// TIA Portal project "TIA_project" (V17)

(* hardware
DEVICE "S71500/ET200MP station_1"  S7-1500 station
   slot 0: "Rail_0"  Rack  6ES7 590-1***0-0AA0
   slot 1: "PLC_1"  CPU 1512C-1 PN  6ES7 512-1CK00-0AB0  V2.1
      slot 3: "CPU display_1"  6ES7591-1AA00-0AA0
DEVICE "HMI_1"  TP700 Comfort
   slot 0: "TP700 Comfort"  TP700 Comfort  6AV2 124-0GC01-0AX0  14.0.1.0
   slot 1: "HMI_RT_1"  TP700 Comfort  6AV2 124-0GC01-0AX0  14.0.1.0
   slot 5: "HMI_1.IE_CP_1"  PROFINET Interface  14.0.1.0
      slot 1: "PROFINET Interface_1"  PROFINET Interface
         slot 1: "Port_1"  Port
         slot 2: "Port_2"  Port
   slot 7: "HMI_1.MPI/DP_CP_1"  MPI/DP Interface  14.0.1.0
*)

// ===== PLC "PLC_1"  CPU 1512C-1 PN =====

VAR_GLOBAL   // PLC tag table "Default tag table"
   "System_Byte" AT %MB1 : Byte;
   "FirstScan" AT %M1.0 : Bool;
   "DiagStatusUpdate" AT %M1.1 : Bool;
   "AlwaysTRUE" AT %M1.2 : Bool;
   "AlwaysFALSE" AT %M1.3 : Bool;
   "Clock_Byte" AT %MB0 : Byte;
   "Clock_10Hz" AT %M0.0 : Bool;
   "Clock_5Hz" AT %M0.1 : Bool;
   "Clock_2.5Hz" AT %M0.2 : Bool;
   "Clock_2Hz" AT %M0.3 : Bool;
   "Clock_1.25Hz" AT %M0.4 : Bool;
   "Clock_1Hz" AT %M0.5 : Bool;
   "Clock_0.625Hz" AT %M0.6 : Bool;
   "Clock_0.5Hz" AT %M0.7 : Bool;
END_VAR

VAR_GLOBAL   // PLC tag table "IO"
   "diVlaveFill_Open" AT %I320.0 : Bool;
   "diVlaveFill_Close" AT %I320.1 : Bool;
   "diVlaveFill_Error" AT %I320.2 : Bool;
   "diVlaveDrain_Open" AT %I320.3 : Bool;
   "diVlaveDrain_Close" AT %I320.4 : Bool;
   "diVlaveDrain_Error" AT %I320.5 : Bool;
   "diMixer_Run" AT %I320.6 : Bool;
   "diMixer_Error" AT %I320.7 : Bool;
   "doValveFill_Open" AT %Q360.0 : Bool;
   "doValveFill_Close" AT %Q360.1 : Bool;
   "doValveDrain_Open" AT %Q360.2 : Bool;
   "doValveDrain_Close" AT %Q360.3 : Bool;
   "doMixer_Run" AT %Q360.4 : Bool;
   "aiWaterLevel" AT %IW340 : Int;
   "aoHeatPower" AT %QW380 : Int;
   "doHeatingEnable" AT %Q360.5 : Bool;
   "aiWaterTemp" AT %IW342 : Int;
END_VAR

// folder: MAUP

TYPE "Valve"
   STRUCT
      State : Struct
         Open : Bool;
         Closed : Bool;
         OpenOut : Bool;
         CloseOut : Bool;
         Err : Bool;
         StartUpFail : Bool;
         AutCtrl : Bool;
         ManCtrl : Bool;
         MayRun : Bool;
         MayAutoRun : Bool;
         GenErr : Bool;
         StColor : Int;
      END_STRUCT;
      Cmd : Struct
         AutCtrl : Bool;
         ManCtrl : Bool;
         OpenMan : Bool;
         StopMan : Bool;
         CloseMan : Bool;
         Req2OpenAut : Bool;
         Req2CloseAut : Bool;
         ResetSUF : Bool;
      END_STRUCT;
      Param : Struct
         Time2Open : Time := t#3s;
      END_STRUCT;
   END_STRUCT;
END_TYPE

TYPE "Engine"
   STRUCT
      State : Struct
         RT : DInt;
         Run : Bool;
         RunOut : Bool;
         Err : Bool;
         StartUpFail : Bool;
         AutCtrl : Bool;
         ManCtrl : Bool;
         MayRun : Bool;
         MayAutoRun : Bool;
         GenErr : Bool;
         StateInt : Int;
      END_STRUCT;
      Cmd : Struct
         SetRT : DInt := -1;
         AutCtrl : Bool;
         ManCtrl : Bool;
         TurnOnMan : Bool;
         TurnOffMan : Bool;
         Req2RunAutCtrl : Bool;
         ResetSUF : Bool;
      END_STRUCT;
      Param : Struct
         Time2Start : Time := T#3s;
      END_STRUCT;
   END_STRUCT;
END_TYPE

TYPE "Tank"
   STRUCT
      ValveFill : "Valve";
      ValveDrain : "Valve";
      Mixer : "Engine";
      Heater : "Heater";
      Draining : "PhaseDraining";
      Filling : "PhaseFilling";
      Heating : "PhaseHeating";
      Mixing : "PhaseMixing";
      GlobalError : Bool;
      WaterTemp : "AI";
      WaterLevel : "AI";
   END_STRUCT;
END_TYPE

TYPE "PhaseMixing"
   STRUCT
      Cmd : Struct
         StartAut : Bool;
         StopAut : Bool;
         StartMan : Bool;
         StopMan : Bool;
         PauseMan : Bool;
         ResumeMan : Bool;
         ResetDone : Bool;
         AutCtrl : Bool;
         ManCtrl : Bool;
      END_STRUCT;
      State : Struct
         Running : Bool;
         Idle : Bool;
         Paused : Bool;
         Done : Bool;
         AutCtrl : Bool;
         ManCtrl : Bool;
         StateInt : Int;
      END_STRUCT;
      Param : Struct
         TimeSec : Int;
      END_STRUCT;
   END_STRUCT;
END_TYPE

TYPE "PhaseFilling"
   STRUCT
      Cmd : Struct
         StartAut : Bool;
         StopAut : Bool;
         StartMan : Bool;
         StopMan : Bool;
         PauseMan : Bool;
         ResumeMan : Bool;
         ResetDone : Bool;
         AutCtrl : Bool;
         ManCtrl : Bool;
      END_STRUCT;
      State : Struct
         Running : Bool;
         Idle : Bool;
         Paused : Bool;
         Done : Bool;
         AutCtrl : Bool;
         ManCtrl : Bool;
         Stateint : Int;
      END_STRUCT;
      Param : Struct
         FillLevel : Real;
      END_STRUCT;
      WaterLevel : Real;
   END_STRUCT;
END_TYPE

TYPE "PhaseDraining"
   STRUCT
      Cmd : Struct
         StartAut : Bool;
         StopAut : Bool;
         StartMan : Bool;
         StopMan : Bool;
         PauseMan : Bool;
         ResumeMan : Bool;
         ResetDone : Bool;
         AutCtrl : Bool;
         ManCtrl : Bool;
      END_STRUCT;
      State : Struct
         Running : Bool;
         Idle : Bool;
         Paused : Bool;
         Done : Bool;
         AutCtrl : Bool;
         ManCtrl : Bool;
         StateInt : Int;
      END_STRUCT;
      Param : Struct
         DrainLevel : Real;
      END_STRUCT;
      WaterLevel : Real;
   END_STRUCT;
END_TYPE

TYPE "PhaseHeating"
   STRUCT
      Cmd : Struct
         StartAut : Bool;
         StopAut : Bool;
         StartMan : Bool;
         StopMan : Bool;
         PauseMan : Bool;
         ResumeMan : Bool;
         ResetDone : Bool;
         AutCtrl : Bool;
         ManCtrl : Bool;
      END_STRUCT;
      State : Struct
         Running : Bool;
         Idle : Bool;
         Paused : Bool;
         Done : Bool;
         AutCtrl : Bool;
         ManCtrl : Bool;
         StateInt : Int;
      END_STRUCT;
      Param : Struct
         ReqTemp : Real;
      END_STRUCT;
      WaterTemp : Real;
   END_STRUCT;
END_TYPE

TYPE "AI"
   STRUCT
      AIScaled : Real;
      TransducerLoLevel : Int;
      TransducerHiLevel : Int := 27648;
      ScaledValLoLevel : Real;
      ScaledValHiLevel : Real := 100.0;
   END_STRUCT;
END_TYPE

TYPE "Heater"
   STRUCT
      State : Struct
         EnableOut : Bool;
         HeatingOut : Real;
         AutCtrl : Bool;
         ManCtrl : Bool;
         StateInt : Int;
      END_STRUCT;
      Cmd : Struct
         AutCtrl : Bool;
         ManCtrl : Bool;
         TurnOnMan : Bool;
         TurnOffMan : Bool;
         Req2RunAutCtrl : Bool;
      END_STRUCT;
      Param : Struct
         HeatingPowerManual : Real;
         HeatingSetPointAutomat : Real;
      END_STRUCT;
   END_STRUCT;
END_TYPE

TYPE "ProcessControl"
   STRUCT
      Cmd : Struct
         Stop : Bool;
         Start : Bool;
      END_STRUCT;
      State : Struct
         Phase : Int;
      END_STRUCT;
   END_STRUCT;
END_TYPE

// folder: (top level)

DATA_BLOCK "ProcessControlFC_DB"   // DB2
{ S7_Optimized_Access := 'TRUE' }
VERSION : 0.1
// stored: InstanceOfName ProcessControlFC
"ProcessControlFC"
BEGIN
END_DATA_BLOCK

DATA_BLOCK "TankFC_DB"   // DB4
{ S7_Optimized_Access := 'TRUE' }
VERSION : 0.1
// stored: InstanceOfName TankFC
"TankFC"
BEGIN
END_DATA_BLOCK

// folder: DBs

DATA_BLOCK "Data"   // DB1
{ S7_Optimized_Access := 'TRUE' }
VERSION : 0.1
   VAR
      ProcessControl1 : "ProcessControl";
      Tank1 : "Tank";
   END_VAR
BEGIN
   Tank1.Filling.Param.FillLevel := 1.5;
   Tank1.ValveDrain.Param.Time2Open := T#30m;
   Tank1.ValveFill.Param.Time2Open := T#30m;
   Tank1.Mixer.Param.Time2Start := T#30m;
   Tank1.WaterTemp.ScaledValLoLevel := 0.0;
   Tank1.WaterTemp.ScaledValHiLevel := 100.0;
   Tank1.WaterLevel.ScaledValHiLevel := 2.0;
   Tank1.Mixing.Param.TimeSec := 15;
   Tank1.Heating.Param.ReqTemp := 60.0;
   Tank1.Heater.Param.HeatingSetPointAutomat := 60.0;
END_DATA_BLOCK

// folder: (top level)

FUNCTION_BLOCK "TankFC"   // FB3, LAD
{ S7_Optimized_Access := 'TRUE' }
VERSION : 0.1
   VAR_INPUT
      diMixer_Running : Bool;
      diMixer_Error : Bool;
      diValveFill_Open : Bool;
      diValveFill_Close : Bool;
      diValveFill_Error : Bool;
      diValveDrain_Open : Bool;
      diValveDrain_Close : Bool;
      diValveDrain_Error : Bool;
      aiWaterLevel : Int;
      aiWaterTemp : Int;
   END_VAR
   VAR_OUTPUT
      doMixerStart : Bool;
      doValveFill_Open : Bool;
      doValveFill_Close : Bool;
      doValveDrain_Open : Bool;
      doValveDrain_Close : Bool;
      doHeatingEnable : Bool;
      aoReqPowerOfHeating : Word;
   END_VAR
   VAR_IN_OUT
      Tank : "Tank";
   END_VAR
   VAR
      Mixer : "Eng_1DO";
      ValveFill : "Val_2DO";
      ValveDrain : "Val_2DO";
      DrainingFC_Instance : "DrainingFC";
      FillingFC_Instance : "FillingFC";
      MixingFC_Instance : "MixingFC";
      Real2AnalogValue_Instance : "Real2AnalogValue";
      HeatingFC_Instance : "HeatingFC";
      HeaterFC_Instance : "HeaterFC";
   END_VAR
   VAR_TEMP
      HeaterReqPower : Real;
   END_VAR
   VAR_TEMP   // added for the SCL form of the ladder/FBD networks
      _w1 : Bool;
      _w2 : Bool;
   END_VAR
BEGIN

REGION Network 1
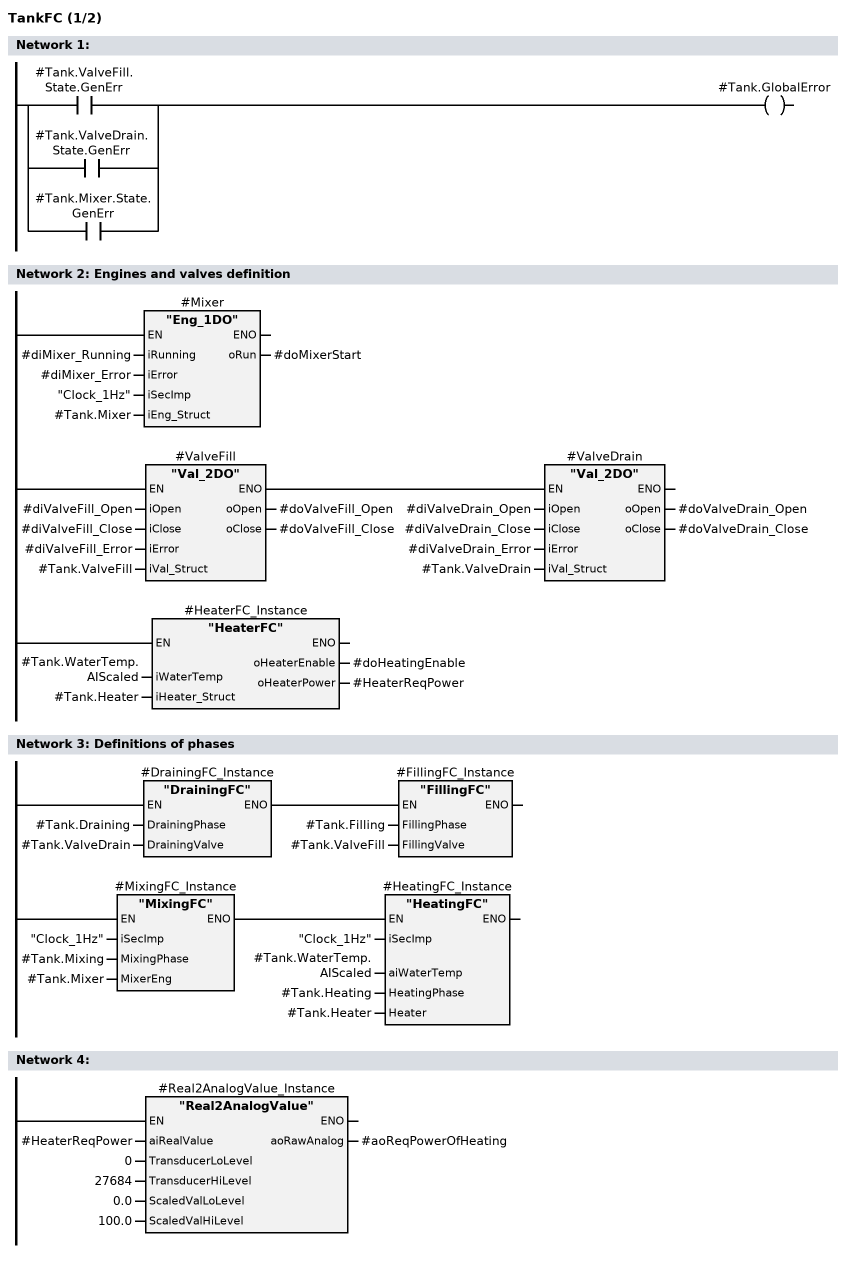
   RUNG wire#powerrail
      Contact( #Tank.ValveFill.State.GenErr )
      wire#w1
      Coil( #Tank.GlobalError )
   END_RUNG
   RUNG wire#powerrail
      Contact( #Tank.ValveDrain.State.GenErr )
   END_RUNG wire#w1
   RUNG wire#powerrail
      Contact( #Tank.Mixer.State.GenErr )
   END_RUNG wire#w1
   // the same network as SCL:
   #Tank.GlobalError := #Tank.ValveFill.State.GenErr OR #Tank.ValveDrain.State.GenErr OR #Tank.Mixer.State.GenErr;
END_REGION

REGION Network 2: Engines and valves definition
   RUNG wire#powerrail
      #Mixer(iRunning := #diMixer_Running, iError := #diMixer_Error, iSecImp := "Clock_1Hz", iEng_Struct := #Tank.Mixer, oRun => #doMixerStart)
   END_RUNG
   RUNG wire#powerrail
      #ValveFill(iOpen := #diValveFill_Open, iClose := #diValveFill_Close, iError := #diValveFill_Error, iVal_Struct := #Tank.ValveFill, oOpen => #doValveFill_Open, oClose => #doValveFill_Close)
      #ValveDrain(iOpen := #diValveDrain_Open, iClose := #diValveDrain_Close, iError := #diValveDrain_Error, iVal_Struct := #Tank.ValveDrain, oOpen => #doValveDrain_Open, oClose => #doValveDrain_Close)
   END_RUNG
   RUNG wire#powerrail
      #HeaterFC_Instance(iWaterTemp := #Tank.WaterTemp.AIScaled, iHeater_Struct := #Tank.Heater, oHeaterEnable => #doHeatingEnable, oHeaterPower => #HeaterReqPower)
   END_RUNG
   // the same network as SCL:
   #Mixer(iRunning := #diMixer_Running,   // "Eng_1DO"
          iError := #diMixer_Error,
          iSecImp := "Clock_1Hz",
          iEng_Struct := #Tank.Mixer,
          oRun => #doMixerStart);
   #ValveFill(iOpen := #diValveFill_Open,   // "Val_2DO"
              iClose := #diValveFill_Close,
              iError := #diValveFill_Error,
              iVal_Struct := #Tank.ValveFill,
              oOpen => #doValveFill_Open,
              oClose => #doValveFill_Close,
              ENO => #_w1);
   IF #_w1 THEN
       #ValveDrain(iOpen := #diValveDrain_Open,   // "Val_2DO"
                   iClose := #diValveDrain_Close,
                   iError := #diValveDrain_Error,
                   iVal_Struct := #Tank.ValveDrain,
                   oOpen => #doValveDrain_Open,
                   oClose => #doValveDrain_Close);
   END_IF;
   #HeaterFC_Instance(iWaterTemp := #Tank.WaterTemp.AIScaled,   // "HeaterFC"
                      iHeater_Struct := #Tank.Heater,
                      oHeaterEnable => #doHeatingEnable,
                      oHeaterPower => #HeaterReqPower);
END_REGION

REGION Network 3: Definitions of phases
   RUNG wire#powerrail
      #DrainingFC_Instance(DrainingPhase := #Tank.Draining, DrainingValve := #Tank.ValveDrain)
      #FillingFC_Instance(FillingPhase := #Tank.Filling, FillingValve := #Tank.ValveFill)
   END_RUNG
   RUNG wire#powerrail
      #MixingFC_Instance(iSecImp := "Clock_1Hz", MixingPhase := #Tank.Mixing, MixerEng := #Tank.Mixer)
      #HeatingFC_Instance(iSecImp := "Clock_1Hz", aiWaterTemp := #Tank.WaterTemp.AIScaled, HeatingPhase := #Tank.Heating, Heater := #Tank.Heater)
   END_RUNG
   // the same network as SCL:
   #DrainingFC_Instance(DrainingPhase := #Tank.Draining, DrainingValve := #Tank.ValveDrain, ENO => #_w1);   // "DrainingFC"
   IF #_w1 THEN
       #FillingFC_Instance(FillingPhase := #Tank.Filling, FillingValve := #Tank.ValveFill);   // "FillingFC"
   END_IF;
   #MixingFC_Instance(iSecImp := "Clock_1Hz", MixingPhase := #Tank.Mixing, MixerEng := #Tank.Mixer, ENO => #_w2);   // "MixingFC"
   IF #_w2 THEN
       #HeatingFC_Instance(iSecImp := "Clock_1Hz",   // "HeatingFC"
                           aiWaterTemp := #Tank.WaterTemp.AIScaled,
                           HeatingPhase := #Tank.Heating,
                           Heater := #Tank.Heater);
   END_IF;
END_REGION

REGION Network 4
   RUNG wire#powerrail
      #Real2AnalogValue_Instance(aiRealValue := #HeaterReqPower, TransducerLoLevel := 0, TransducerHiLevel := 27684, ScaledValLoLevel := 0.0, ScaledValHiLevel := 100.0, aoRawAnalog => #aoReqPowerOfHeating)
   END_RUNG
   // the same network as SCL:
   #Real2AnalogValue_Instance(aiRealValue := #HeaterReqPower,   // "Real2AnalogValue"
                           TransducerLoLevel := 0,
                           TransducerHiLevel := 27684,
                           ScaledValLoLevel := 0.0,
                           ScaledValHiLevel := 100.0,
                           aoRawAnalog => #aoReqPowerOfHeating);
END_REGION

REGION Network 5: Analog scaling
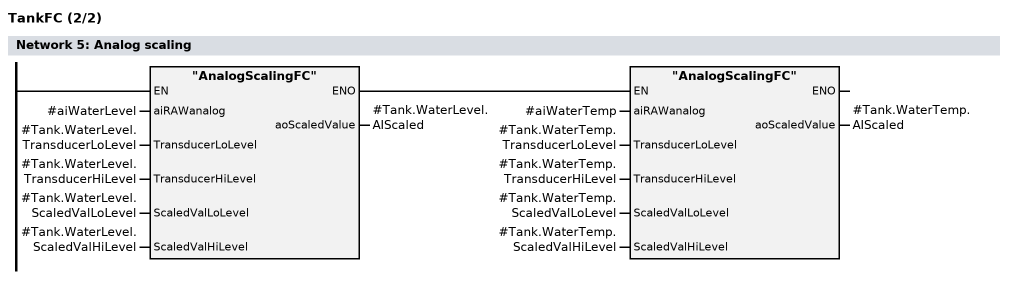
   RUNG wire#powerrail
      "AnalogScalingFC"(aiRAWanalog := #aiWaterLevel, TransducerLoLevel := #Tank.WaterLevel.TransducerLoLevel, TransducerHiLevel := #Tank.WaterLevel.TransducerHiLevel, ScaledValLoLevel := #Tank.WaterLevel.ScaledValLoLevel, ScaledValHiLevel := #Tank.WaterLevel.ScaledValHiLevel, aoScaledValue => #Tank.WaterLevel.AIScaled)
      "AnalogScalingFC"(aiRAWanalog := #aiWaterTemp, TransducerLoLevel := #Tank.WaterTemp.TransducerLoLevel, TransducerHiLevel := #Tank.WaterTemp.TransducerHiLevel, ScaledValLoLevel := #Tank.WaterTemp.ScaledValLoLevel, ScaledValHiLevel := #Tank.WaterTemp.ScaledValHiLevel, aoScaledValue => #Tank.WaterTemp.AIScaled)
   END_RUNG
   // the same network as SCL:
   "AnalogScalingFC"(aiRAWanalog := #aiWaterLevel,
                     TransducerLoLevel := #Tank.WaterLevel.TransducerLoLevel,
                     TransducerHiLevel := #Tank.WaterLevel.TransducerHiLevel,
                     ScaledValLoLevel := #Tank.WaterLevel.ScaledValLoLevel,
                     ScaledValHiLevel := #Tank.WaterLevel.ScaledValHiLevel,
                     aoScaledValue => #Tank.WaterLevel.AIScaled,
                     ENO => #_w1);
   IF #_w1 THEN
       "AnalogScalingFC"(aiRAWanalog := #aiWaterTemp,
                         TransducerLoLevel := #Tank.WaterTemp.TransducerLoLevel,
                         TransducerHiLevel := #Tank.WaterTemp.TransducerHiLevel,
                         ScaledValLoLevel := #Tank.WaterTemp.ScaledValLoLevel,
                         ScaledValHiLevel := #Tank.WaterTemp.ScaledValHiLevel,
                         aoScaledValue => #Tank.WaterTemp.AIScaled);
   END_IF;
END_REGION

REGION Network 6 (SCL): Data transfer
   #Tank.Draining.WaterLevel := #Tank.WaterLevel.AIScaled;
   #Tank.Filling.WaterLevel := #Tank.WaterLevel.AIScaled;
   #Tank.Heating.WaterTemp := #Tank.WaterTemp.AIScaled;
END_REGION
END_FUNCTION_BLOCK

FUNCTION_BLOCK "ProcessControlFC"   // FB10, SCL
{ S7_Optimized_Access := 'TRUE' }
VERSION : 0.1
   VAR_IN_OUT
      Tank : "Tank";
      ProcessControl : "ProcessControl";
   END_VAR
   VAR CONSTANT
      StateIdle : Int := 0;
      StateFilling : Int := 1;
      StateFilled : Int := 2;
      StateHeating : Int := 3;
      StateHeated : Int := 4;
      StateMixing : Int := 5;
      StateMixed : Int := 6;
      StateDraining : Int := 7;
   END_VAR
BEGIN
   CASE #ProcessControl.State.Phase OF
       #StateIdle:
           IF #Tank.Filling.State.Running THEN
               #ProcessControl.State.Phase := #StateFilling;
           END_IF;
       #StateFilling:
           IF #Tank.Filling.State.Done THEN
               #ProcessControl.State.Phase := #StateFilled;
           END_IF;
       #StateFilled:
           #Tank.Heater.Param.HeatingSetPointAutomat := 60;
           #Tank.Mixing.Param.TimeSec := -1;
           #Tank.Heating.Cmd.StartAut := TRUE;
           #Tank.Mixing.Cmd.StartAut := TRUE;
           IF #Tank.Heating.State.Running AND #Tank.Mixing.State.Running THEN
               #ProcessControl.State.Phase := #StateHeating;
           END_IF;
       #StateHeating:
           IF #Tank.Heating.State.Done THEN
               #ProcessControl.State.Phase := #StateHeated;
           END_IF;
       #StateHeated:
           #Tank.Mixing.Param.TimeSec := 30;
           #Tank.Mixing.Cmd.StartAut := TRUE;
           IF #Tank.Mixing.State.Running THEN
               #ProcessControl.State.Phase := #StateMixing;
           END_IF;
       #StateMixing:
           IF #Tank.Mixing.State.Done THEN
               #ProcessControl.State.Phase := #StateMixed;
               #Tank.Heating.Cmd.StopAut := TRUE;
           END_IF;
       #StateMixed:
           #Tank.Draining.Param.DrainLevel := 0;
           #Tank.Draining.Cmd.StartAut := TRUE;
           IF #Tank.Draining.State.Running THEN
               #ProcessControl.State.Phase := #StateDraining;
           END_IF;
       #StateDraining:
           IF #Tank.Draining.#State.Done THEN
               #ProcessControl.State.Phase := #StateIdle;
           END_IF;
   END_CASE;

   IF #ProcessControl.Cmd.Start THEN
       IF #ProcessControl.State.Phase = #StateIdle THEN
           #Tank.Filling.Param.FillLevel := 1.5;
           #Tank.Filling.Cmd.StartAut := TRUE;
       END_IF;
       #ProcessControl.Cmd.Start := FALSE;
   END_IF;

   IF #ProcessControl.Cmd.Stop THEN
       #Tank.Filling.Cmd.StopAut := TRUE;
       #Tank.Heating.Cmd.StopAut := TRUE;
       #Tank.Mixing.Cmd.StopAut := TRUE;
       #Tank.Draining.Cmd.StopAut := TRUE;
       #ProcessControl.State.Phase := #StateIdle;
       #ProcessControl.Cmd.Stop := FALSE;
   END_IF;
END_FUNCTION_BLOCK

ORGANIZATION_BLOCK "Main"   // OB1, LAD, ProgramCycle
TITLE = "Main Program Sweep (Cycle)"
{ S7_Optimized_Access := 'TRUE' }
VERSION : 0.1
   VAR_INPUT
      Initial_Call : Bool;   // Initial call of this OB
      Remanence : Bool;   // =True, if remanent data are available
   END_VAR
BEGIN
END_ORGANIZATION_BLOCK

ORGANIZATION_BLOCK "Cyclic interrupt10ms"   // OB31, LAD, CyclicInterrupt
{ S7_Optimized_Access := 'TRUE' }
VERSION : 0.1
   VAR_INPUT
      Initial_Call : Bool;   // Initial call of this OB
      Event_Count : Int;   // Events discarded
   END_VAR
BEGIN

REGION Network 1
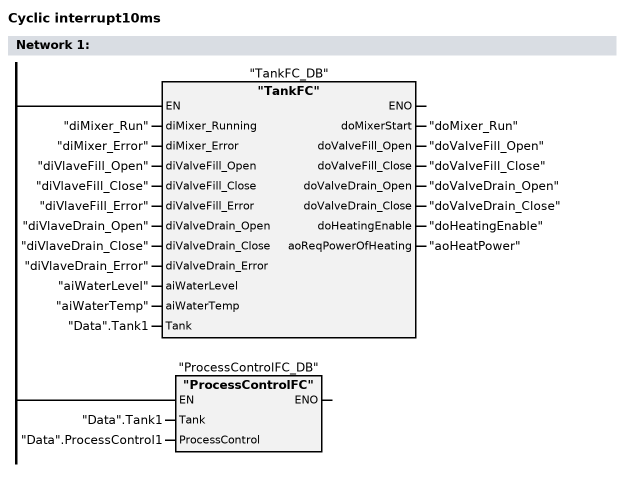
   RUNG wire#powerrail
      "TankFC_DB"(diMixer_Running := "diMixer_Run", diMixer_Error := "diMixer_Error", diValveFill_Open := "diVlaveFill_Open", diValveFill_Close := "diVlaveFill_Close", diValveFill_Error := "diVlaveFill_Error", diValveDrain_Open := "diVlaveDrain_Open", diValveDrain_Close := "diVlaveDrain_Close", diValveDrain_Error := "diVlaveDrain_Error", aiWaterLevel := "aiWaterLevel", aiWaterTemp := "aiWaterTemp", Tank := "Data".Tank1, doMixerStart => "doMixer_Run", doValveFill_Open => "doValveFill_Open", doValveFill_Close => "doValveFill_Close", doValveDrain_Open => "doValveDrain_Open", doValveDrain_Close => "doValveDrain_Close", doHeatingEnable => "doHeatingEnable", aoReqPowerOfHeating => "aoHeatPower")
   END_RUNG
   RUNG wire#powerrail
      "ProcessControlFC_DB"(Tank := "Data".Tank1, ProcessControl := "Data".ProcessControl1)
   END_RUNG
   // the same network as SCL:
   "TankFC_DB"(diMixer_Running := "diMixer_Run",   // "TankFC"
               diMixer_Error := "diMixer_Error",
               diValveFill_Open := "diVlaveFill_Open",
               diValveFill_Close := "diVlaveFill_Close",
               diValveFill_Error := "diVlaveFill_Error",
               diValveDrain_Open := "diVlaveDrain_Open",
               diValveDrain_Close := "diVlaveDrain_Close",
               diValveDrain_Error := "diVlaveDrain_Error",
               aiWaterLevel := "aiWaterLevel",
               aiWaterTemp := "aiWaterTemp",
               Tank := "Data".Tank1,
               doMixerStart => "doMixer_Run",
               doValveFill_Open => "doValveFill_Open",
               doValveFill_Close => "doValveFill_Close",
               doValveDrain_Open => "doValveDrain_Open",
               doValveDrain_Close => "doValveDrain_Close",
               doHeatingEnable => "doHeatingEnable",
               aoReqPowerOfHeating => "aoHeatPower");
   "ProcessControlFC_DB"(Tank := "Data".Tank1, ProcessControl := "Data".ProcessControl1);   // "ProcessControlFC"
END_REGION
END_ORGANIZATION_BLOCK

ORGANIZATION_BLOCK "Startup"   // OB100, SCL, Startup
TITLE = "Complete Restart"
{ S7_Optimized_Access := 'TRUE' }
VERSION : 0.1
   VAR_INPUT
      LostRetentive : Bool;   // True if retentive data are lost
      LostRTC : Bool;   // True if date and time are lost
   END_VAR
BEGIN
END_ORGANIZATION_BLOCK

// folder: FCs

FUNCTION_BLOCK "Eng_1DO"   // FB1, SCL
{ S7_Optimized_Access := 'TRUE' }
VERSION : 0.1
   VAR_INPUT
      iRunning : Bool;
      iError : Bool;
      iSecImp : Bool;
   END_VAR
   VAR_OUTPUT
      oRun : Bool;
   END_VAR
   VAR_IN_OUT
      iEng_Struct : "Engine";
   END_VAR
   VAR
      SecImpEdge : R_TRIG;
      SUF_Timer : TON_TIME;
   END_VAR
   VAR CONSTANT
      Running : Int := 0;
      Stop : Int := 1;
      RunningAndErr : Int := 2;
      Err : Int := 3;
   END_VAR
BEGIN
   REGION RunningTime
       // counting running time of engine - (motoseconds in real situation it should be moto hours)
       // detection rising edge of input secimp - should be conected 1Hz internal clock from PLC

       #SecImpEdge(CLK := #iSecImp);
       IF #SecImpEdge.Q AND #iRunning THEN
           #iEng_Struct.State.RT += 1;
       END_IF;

       IF #iEng_Struct.Cmd.SetRT >= 0 THEN
           #iEng_Struct.State.RT := #iEng_Struct.Cmd.SetRT;
           #iEng_Struct.Cmd.SetRT := -1;
       END_IF;
   END_REGION

   REGION RunState 
       // set real state of engine input into engine structure - input of running
       // engine can be taken from frequential converter, speed sensor, or just
       // from switching element

       #iEng_Struct.State.Run := #iRunning;
   END_REGION

   REGION Manual/Automat 
       // switching state of engine - automatic or manual control (default state is manual)

       IF (#iEng_Struct.Cmd.AutCtrl AND #iEng_Struct.Cmd.ManCtrl) OR (NOT #iEng_Struct.State.AutCtrl AND NOT #iEng_Struct.State.ManCtrl) THEN
           #iEng_Struct.State.AutCtrl := FALSE;
           #iEng_Struct.State.ManCtrl := TRUE;
       ELSIF #iEng_Struct.Cmd.AutCtrl THEN
           #iEng_Struct.State.AutCtrl := TRUE;
           #iEng_Struct.State.ManCtrl := FALSE;
       ELSIF #iEng_Struct.Cmd.ManCtrl THEN
           #iEng_Struct.State.AutCtrl := FALSE;
           #iEng_Struct.State.ManCtrl := TRUE;
       END_IF;

       #iEng_Struct.Cmd.AutCtrl := FALSE;
       #iEng_Struct.Cmd.ManCtrl := FALSE;
   END_REGION

   REGION MR/MAR 
       // setting auxilary signals (may run, may auto run) - MR AND NOT MAR - eng should be started in manual mode,
       // MAR - should be started in automatic mode

       #iEng_Struct.State.MayRun := #iEng_Struct.State.ManCtrl AND NOT #iEng_Struct.State.Err;
       #iEng_Struct.State.MayAutoRun := #iEng_Struct.State.AutCtrl AND NOT #iEng_Struct.State.Err;
   END_REGION

   REGION ManCtrl
       // processing manual actions - if command is processed, it is set to FALSE even if can't be processed
       // Engine commands are turn off (stop) and turn on (start)

       IF #iEng_Struct.Cmd.TurnOnMan AND #iEng_Struct.State.MayRun THEN
           #iEng_Struct.State.RunOut := TRUE;
       END_IF;

       IF #iEng_Struct.Cmd.TurnOffMan AND #iEng_Struct.State.MayRun THEN
           #iEng_Struct.State.RunOut := FALSE;
       END_IF;

       #iEng_Struct.Cmd.TurnOnMan := FALSE;
       #iEng_Struct.Cmd.TurnOffMan := FALSE;
   END_REGION

   REGION AutCtrl 
       //if request to run in automatic mode set outputs to right states if MAR
       //AutoRequest shouldn't be reseted to false state

       IF  #iEng_Struct.State.MayAutoRun THEN
           #iEng_Struct.State.RunOut := #iEng_Struct.Cmd.Req2RunAutCtrl;
       END_IF;
   END_REGION

   REGION ErrStates
       // definition of error states 
       // error - input from digital input of plc - fyzical state of engine 
       // calculating start up fail - if output is sets to start engine, it's expected feedback from running signal in defined time, if feedback doesn't show in this time, it should be start up fail error
       // merge of these two error is general error

       #SUF_Timer(IN := #iEng_Struct.State.RunOut,
                  PT := #iEng_Struct.Param.Time2Start);
       IF #SUF_Timer.Q AND NOT #iRunning THEN
           #iEng_Struct.State.StartUpFail := TRUE;
       END_IF;

       #iEng_Struct.State.Err := #iError;

       #iEng_Struct.State.GenErr := #iEng_Struct.State.StartUpFail OR #iEng_Struct.State.Err;

       IF #iEng_Struct.Cmd.ResetSUF THEN
           #iEng_Struct.State.StartUpFail := FALSE;
       END_IF;
       #iEng_Struct.Cmd.ResetSUF := FALSE;

       IF #iEng_Struct.State.GenErr THEN
           #iEng_Struct.State.RunOut := FALSE;
       END_IF;
   END_REGION

   #oRun := #iEng_Struct.State.RunOut;

   REGION StatusInt
       //write combination of states into int value for visualization (engine - combination of running state and error)

       IF NOT #iEng_Struct.State.GenErr THEN
           IF #iEng_Struct.State.Run THEN
               #iEng_Struct.State.StateInt := #Running;
           ELSE
               #iEng_Struct.State.StateInt := #Stop;
           END_IF;
       ELSE
           IF #iEng_Struct.State.Run THEN
               #iEng_Struct.State.StateInt := #RunningAndErr;
           ELSE
               #iEng_Struct.State.StateInt := #Err;
           END_IF;
       END_IF;
   END_REGION
END_FUNCTION_BLOCK

FUNCTION_BLOCK "Val_2DO"   // FB2, SCL
{ S7_Optimized_Access := 'TRUE' }
VERSION : 0.1
   VAR_INPUT
      iOpen : Bool;
      iClose : Bool;
      iError : Bool;
   END_VAR
   VAR_OUTPUT
      oOpen : Bool;
      oClose : Bool;
   END_VAR
   VAR_IN_OUT
      iVal_Struct : "Valve";
   END_VAR
   VAR
      fTimeToOpen : TON_TIME;
      fTimeToClose : TON_TIME;
   END_VAR
   VAR CONSTANT
      Open : Int := 0;
      Closed : Int := 1;
      OpenAndErr : Int := 2;
      ClosedAndErr : Int := 3;
      NotOpenNotClosedNotErr : Int := 4;
      NotOpenNotClosedAndErr : Int := 5;
      OpenAndClosedAndErr : Int := 6;
      OpenAndClosedNotErr : Int := 7;
   END_VAR
BEGIN
   REGION OpenState 
       // set real state of valve input into valve structure - input of valve can be taken from limit sensor...
       // input - open?
       #iVal_Struct.State.Open := #iOpen;
       // input - closed?
       #iVal_Struct.State.Closed := #iClose;
   END_REGION

   REGION Manual/Automat
       // switching state of engine - automatic or manual control (default state is manual)
       IF (#iVal_Struct.Cmd.AutCtrl AND #iVal_Struct.Cmd.ManCtrl) OR (NOT #iVal_Struct.State.AutCtrl AND NOT #iVal_Struct.State.ManCtrl) THEN
           #iVal_Struct.State.AutCtrl := FALSE;
           #iVal_Struct.State.ManCtrl := TRUE;
       ELSIF #iVal_Struct.Cmd.AutCtrl THEN
           #iVal_Struct.State.AutCtrl := TRUE;
           #iVal_Struct.State.ManCtrl := FALSE;
       ELSIF #iVal_Struct.Cmd.ManCtrl THEN
           #iVal_Struct.State.AutCtrl := FALSE;
           #iVal_Struct.State.ManCtrl := TRUE;
       END_IF;

       #iVal_Struct.Cmd.AutCtrl := FALSE;
       #iVal_Struct.Cmd.ManCtrl := FALSE;
   END_REGION

   REGION MR/MAR
       // setting auxilary signals (may run, may auto run) - MR AND NOT MAR - eng should be started in manual mode, MAR - should be started in automatic mode

       #iVal_Struct.State.MayRun := #iVal_Struct.State.ManCtrl AND NOT #iVal_Struct.State.Err;
       #iVal_Struct.State.MayAutoRun := #iVal_Struct.State.AutCtrl AND NOT #iVal_Struct.State.Err;
   END_REGION

   REGION ManCtrl
       // processing manual actions - if command is processed, it is sets to FALSE even if can't be processed
       // Valve commands are open, close and stop - valve can be stopped intermediate position

       // Open control
       IF #iVal_Struct.Cmd.OpenMan AND #iVal_Struct.State.MayRun THEN
           #iVal_Struct.State.CloseOut := FALSE;
           #iVal_Struct.State.OpenOut := TRUE;
       END_IF;

       // Close control
       IF #iVal_Struct.Cmd.CloseMan AND #iVal_Struct.State.MayRun THEN
           #iVal_Struct.State.OpenOut := FALSE;
           #iVal_Struct.State.CloseOut := TRUE;
       END_IF;

       // stop control
       IF #iVal_Struct.Cmd.StopMan AND #iVal_Struct.State.MayRun THEN
           #iVal_Struct.State.OpenOut := FALSE;
           #iVal_Struct.State.CloseOut := FALSE;
       END_IF;

       // clear commands
       #iVal_Struct.Cmd.OpenMan := FALSE;
       #iVal_Struct.Cmd.StopMan := FALSE;
       #iVal_Struct.Cmd.CloseMan := FALSE;
   END_REGION

   REGION AutCtrl
       //if request to run in automatic mode -> set outputs to right states if MAR
       //AutoRequest shouldn't be reseted to false state
       //if request to open and request to close are setted to 1 simultaneously - outputs should be 0.

       IF #iVal_Struct.State.MayAutoRun THEN
           IF (#iVal_Struct.Cmd.Req2OpenAut AND NOT #iVal_Struct.Cmd.Req2CloseAut) THEN
               #iVal_Struct.State.CloseOut := FALSE;
               #iVal_Struct.State.OpenOut := TRUE;
           ELSIF (NOT #iVal_Struct.Cmd.Req2OpenAut AND #iVal_Struct.Cmd.Req2CloseAut) THEN
               #iVal_Struct.State.OpenOut := FALSE;
               #iVal_Struct.State.CloseOut := TRUE;
           ELSE // simultanesly activated or deactivated
               #iVal_Struct.State.OpenOut := FALSE;
               #iVal_Struct.State.CloseOut := FALSE;
           END_IF;
       END_IF;

   END_REGION

   REGION ErrStates
       // definition of error states 
       // error - input from digital input of plc - fyzical state of valve
       // calculating start up fail - if output is sets to open or close, it's expected feedback from limit sensor in defined time, if feedback doesn't show in this time, it should be start up fail error
       // merge of these two error is general error
       // error is both inputs (open and closed) true state

       #fTimeToOpen(IN := #iVal_Struct.State.OpenOut AND NOT #iVal_Struct.State.CloseOut,
                    PT := #iVal_Struct.Param.Time2Open);
       #fTimeToClose(IN := NOT #iVal_Struct.State.OpenOut AND #iVal_Struct.State.CloseOut,
                     PT := #iVal_Struct.Param.Time2Open);

       IF (#fTimeToOpen.Q AND NOT #iOpen) OR (#fTimeToClose.Q AND NOT #iClose) THEN
           #iVal_Struct.State.StartUpFail := TRUE;
       END_IF;

       // set the input Error to state 
       #iVal_Struct.State.Err := #iError;

       // Merge the errors
       #iVal_Struct.State.GenErr := #iVal_Struct.State.StartUpFail OR #iVal_Struct.State.Err;

       // start up fail can be reseted by operator, command resetSUF, resets SUF and engine should be started again
       IF #iVal_Struct.Cmd.ResetSUF THEN
           #iVal_Struct.State.StartUpFail := FALSE;
       END_IF;
       // reset the command
       #iVal_Struct.Cmd.ResetSUF := FALSE;

       // if error state exists outputs should be in stop state
       IF #iVal_Struct.State.GenErr THEN
           #iVal_Struct.State.OpenOut := FALSE;
           #iVal_Struct.State.CloseOut := FALSE;
       END_IF;

   END_REGION

   #oOpen := #iVal_Struct.State.OpenOut;
   #oClose := #iVal_Struct.State.CloseOut;

   REGION StatusInt
       //write combination of states into int value for visualization (valve - combination of open, close state and error)
       IF #iVal_Struct.State.Open AND NOT #iVal_Struct.State.Closed AND NOT #iVal_Struct.State.GenErr THEN
           #iVal_Struct.State.StColor := #Open;
       ELSIF NOT #iVal_Struct.State.Open AND #iVal_Struct.State.Closed AND NOT #iVal_Struct.State.GenErr THEN
           #iVal_Struct.State.StColor := #Closed;
       ELSIF #iVal_Struct.State.Open AND NOT #iVal_Struct.State.Closed AND #iVal_Struct.State.GenErr THEN
           #iVal_Struct.State.StColor := #OpenAndErr;
       ELSIF NOT #iVal_Struct.State.Open AND #iVal_Struct.State.Closed AND #iVal_Struct.State.GenErr THEN
           #iVal_Struct.State.StColor := #ClosedAndErr;
       ELSIF NOT #iVal_Struct.State.Open AND NOT #iVal_Struct.State.Closed AND NOT #iVal_Struct.State.GenErr THEN
           #iVal_Struct.State.StColor := #NotOpenNotClosedNotErr;
       ELSIF NOT #iVal_Struct.State.Open AND NOT #iVal_Struct.State.Closed AND #iVal_Struct.State.GenErr THEN
           #iVal_Struct.State.StColor := #NotOpenNotClosedAndErr;
       ELSIF #iVal_Struct.State.Open AND #iVal_Struct.State.Closed AND #iVal_Struct.State.GenErr THEN
           #iVal_Struct.State.StColor := #OpenAndClosedAndErr;
       ELSIF #iVal_Struct.State.Open AND #iVal_Struct.State.Closed AND NOT #iVal_Struct.State.GenErr THEN
           #iVal_Struct.State.StColor := #OpenAndClosedNotErr;
       END_IF;
   END_REGION
END_FUNCTION_BLOCK

FUNCTION_BLOCK "FillingFC"   // FB4, SCL
{ S7_Optimized_Access := 'TRUE' }
VERSION : 0.1
   VAR_IN_OUT
      FillingPhase : "PhaseFilling";
      FillingValve : "Valve";
   END_VAR
   VAR CONSTANT
      Idle : Int := 0;
      Running : Int := 1;
      Pause : Int := 2;
   END_VAR
BEGIN
   REGION Aut/Man
       // switching state of engine - automatic or manual control (default state is manual)

       IF (#FillingPhase.Cmd.AutCtrl AND #FillingPhase.Cmd.ManCtrl) OR (NOT #FillingPhase.State.AutCtrl AND NOT #FillingPhase.State.ManCtrl) THEN
           #FillingPhase.State.AutCtrl := FALSE;
           #FillingPhase.State.ManCtrl := TRUE;
       ELSIF #FillingPhase.Cmd.AutCtrl THEN
           #FillingPhase.State.AutCtrl := TRUE;
           #FillingPhase.State.ManCtrl := FALSE;
       ELSIF #FillingPhase.Cmd.ManCtrl THEN
           #FillingPhase.State.AutCtrl := FALSE;
           #FillingPhase.State.ManCtrl := TRUE;
       END_IF;

       #FillingPhase.Cmd.AutCtrl := FALSE;
       #FillingPhase.Cmd.ManCtrl := FALSE;
    END_REGION

   REGION ManCtrl
       // processing manual actions - if command is processed, it is sets to FALSE even if can't be processed
       // Phase commands are start, stop, pause and resume 
       // Start - open filling valve 
       // Stop - close filling valve
       // Pause - close filling valve
       // Resume - open filling valve
       // real states of phase are writed into states in phase structure

       IF #FillingPhase.State.ManCtrl THEN
           IF #FillingPhase.Cmd.StartMan AND #FillingPhase.State.Idle THEN
               #FillingPhase.State.Running := TRUE;
               #FillingPhase.State.Idle := FALSE;
               #FillingPhase.State.Paused := FALSE;
               #FillingPhase.State.Done := FALSE;
           ELSIF #FillingPhase.Cmd.StopMan THEN
               #FillingPhase.State.Running := FALSE;
               #FillingPhase.State.Idle := TRUE;
               #FillingPhase.State.Paused := FALSE;
               #FillingPhase.State.Done := FALSE;
           ELSIF #FillingPhase.Cmd.PauseMan AND #FillingPhase.State.Running THEN
               #FillingPhase.State.Running := FALSE;
               #FillingPhase.State.Idle := FALSE;
               #FillingPhase.State.Paused := TRUE;
               #FillingPhase.State.Done := FALSE;
           ELSIF #FillingPhase.Cmd.ResumeMan AND #FillingPhase.State.Paused THEN
               #FillingPhase.State.Running := TRUE;
               #FillingPhase.State.Idle := FALSE;
               #FillingPhase.State.Paused := FALSE;
               #FillingPhase.State.Done := FALSE;
           END_IF;
       END_IF;

       #FillingPhase.Cmd.StartMan := FALSE;
       #FillingPhase.Cmd.StopMan := FALSE;
       #FillingPhase.Cmd.PauseMan := FALSE;
       #FillingPhase.Cmd.ResumeMan := FALSE;
    END_REGION

   REGION AutCtrl
       // if request to run in automatic mode and phase can be run in automatic mode switch phase to running

       IF #FillingPhase.State.AutCtrl THEN
           IF #FillingPhase.Cmd.StartAut THEN
               #FillingPhase.State.Running := TRUE;
               #FillingPhase.State.Idle := FALSE;
               #FillingPhase.State.Paused := FALSE;
               #FillingPhase.State.Done := FALSE;
           ELSIF #FillingPhase.Cmd.StopAut THEN
               #FillingPhase.State.Running := FALSE;
               #FillingPhase.State.Idle := TRUE;
               #FillingPhase.State.Paused := FALSE;
               #FillingPhase.State.Done := FALSE;
           END_IF;
       END_IF;

       #FillingPhase.Cmd.StartAut := FALSE;
       #FillingPhase.Cmd.StopAut := FALSE;
    END_REGION

   REGION Done
       //every phase should have finish condition - filling phase - if water level is above requested level
       //after that done state should be setted to 1

       IF #FillingPhase.State.Running AND (#FillingPhase.WaterLevel >= #FillingPhase.Param.FillLevel AND NOT (#FillingPhase.WaterLevel = 2.0)) THEN
           #FillingPhase.Cmd.StopAut := TRUE;
           #FillingPhase.Cmd.StopMan := TRUE;
           #FillingPhase.State.Done := TRUE;
       END_IF;

       IF #FillingPhase.State.Paused OR #FillingPhase.State.Idle THEN
           #FillingPhase.State.Done := TRUE;
       END_IF;

       // command reset done resets done state and than resets command

       IF #FillingPhase.Cmd.ResetDone THEN
           #FillingPhase.State.Done := FALSE;
       END_IF;
       #FillingPhase.Cmd.ResetDone := FALSE;
   END_REGION

   REGION States 
       //Command valve in cases of states

       IF #FillingPhase.State.Running THEN
           #FillingValve.Cmd.Req2OpenAut := TRUE;
           #FillingValve.Cmd.Req2CloseAut := FALSE;
       ELSE
           #FillingValve.Cmd.Req2OpenAut := FALSE;
           #FillingValve.Cmd.Req2CloseAut := TRUE;
       END_IF;
   END_REGION

   // delault state of phase - if not any state sets state to idle

   IF NOT #FillingPhase.State.Running AND NOT #FillingPhase.State.Idle AND NOT #FillingPhase.State.Paused THEN
       #FillingPhase.State.Idle := TRUE;
   END_IF;

   // write binary states into int value for visualization

   IF #FillingPhase.State.Running THEN
       #FillingPhase.State.Stateint := #Running;
   ELSIF #FillingPhase.State.Idle THEN
       #FillingPhase.State.Stateint := #Idle;
   ELSE
       #FillingPhase.State.Stateint := #Pause;
   END_IF;
END_FUNCTION_BLOCK

FUNCTION_BLOCK "DrainingFC"   // FB5, SCL
{ S7_Optimized_Access := 'TRUE' }
VERSION : 0.1
   VAR_IN_OUT
      DrainingPhase : "PhaseDraining";
      DrainingValve : "Valve";
   END_VAR
   VAR CONSTANT
      Idle : Int := 0;
      Running : Int := 1;
      Pause : Int := 2;
   END_VAR
BEGIN
   REGION Aut/Man
       // switching state of engine - automatic or manual control (default state is manual)

       IF (#DrainingPhase.Cmd.AutCtrl AND #DrainingPhase.Cmd.ManCtrl) OR (NOT #DrainingPhase.State.AutCtrl AND NOT #DrainingPhase.State.ManCtrl) THEN
           #DrainingPhase.State.AutCtrl := FALSE;
           #DrainingPhase.State.ManCtrl := TRUE;
       ELSIF #DrainingPhase.Cmd.AutCtrl THEN
           #DrainingPhase.State.AutCtrl := TRUE;
           #DrainingPhase.State.ManCtrl := FALSE;
       ELSIF #DrainingPhase.Cmd.ManCtrl THEN
           #DrainingPhase.State.AutCtrl := FALSE;
           #DrainingPhase.State.ManCtrl := TRUE;
       END_IF;

       #DrainingPhase.Cmd.AutCtrl := FALSE;
       #DrainingPhase.Cmd.ManCtrl := FALSE;
   END_REGION

   REGION ManCtrl
       // processing manual actions - if command is processed, it is sets to FALSE even if can't be processed
       // Phase commands are start, stop, pause and resume 
       // Start - open draining valve 
       // Stop - close draining valve
       // Pause - close draining valve
       // Resume - open draining valve
       // real states of phase are writed into states in phase structure

       IF #DrainingPhase.State.ManCtrl THEN
           IF #DrainingPhase.Cmd.StartMan AND #DrainingPhase.State.Idle THEN
               #DrainingPhase.State.Running := TRUE;
               #DrainingPhase.State.Idle := FALSE;
               #DrainingPhase.State.Paused := FALSE;
               #DrainingPhase.State.Done := FALSE;
           ELSIF #DrainingPhase.Cmd.StopMan THEN
               #DrainingPhase.State.Running := FALSE;
               #DrainingPhase.State.Idle := TRUE;
               #DrainingPhase.State.Paused := FALSE;
               #DrainingPhase.State.Done := FALSE;
           ELSIF #DrainingPhase.Cmd.PauseMan AND #DrainingPhase.State.Running THEN
               #DrainingPhase.State.Running := FALSE;
               #DrainingPhase.State.Idle := FALSE;
               #DrainingPhase.State.Paused := TRUE;
               #DrainingPhase.State.Done := FALSE;
           ELSIF #DrainingPhase.Cmd.ResumeMan AND #DrainingPhase.State.Paused THEN
               #DrainingPhase.State.Running := TRUE;
               #DrainingPhase.State.Idle := FALSE;
               #DrainingPhase.State.Paused := FALSE;
               #DrainingPhase.State.Done := FALSE;
           END_IF;
       END_IF;

       #DrainingPhase.Cmd.StartMan := FALSE;
       #DrainingPhase.Cmd.StopMan := FALSE;
       #DrainingPhase.Cmd.PauseMan := FALSE;
       #DrainingPhase.Cmd.ResumeMan := FALSE;
   END_REGION

   REGION AutCtrl
       //if request to run in automatic mode -> set auto request to open of filling valve to 1 and close to 0, if not open 0 close 1
       // commands should be sets to false after their processing

       IF #DrainingPhase.State.AutCtrl THEN
           IF #DrainingPhase.Cmd.StartAut THEN
               #DrainingPhase.State.Running := TRUE;
               #DrainingPhase.State.Idle := FALSE;
               #DrainingPhase.State.Paused := FALSE;
               #DrainingPhase.State.Done := FALSE;
           ELSIF #DrainingPhase.Cmd.StopAut THEN
               #DrainingPhase.State.Running := FALSE;
               #DrainingPhase.State.Idle := TRUE;
               #DrainingPhase.State.Paused := FALSE;
               #DrainingPhase.State.Done := FALSE;
           END_IF;
       END_IF;

       #DrainingPhase.Cmd.StartAut := FALSE;
       #DrainingPhase.Cmd.StopAut := FALSE;
   END_REGION

   REGION Done
       //every phase should have finish condition - draining phase - if water level is below requested level
       //after that done state should be setted to 1

       IF #DrainingPhase.State.Running AND (#DrainingPhase.WaterLevel <= #DrainingPhase.Param.DrainLevel OR #DrainingPhase.WaterLevel = 2.0) THEN
           #DrainingPhase.Cmd.StopAut := TRUE;
           #DrainingPhase.Cmd.StopMan := TRUE;
           #DrainingPhase.State.Done := TRUE;
       END_IF;

       IF #DrainingPhase.State.Paused OR #DrainingPhase.State.Idle THEN
           #DrainingPhase.State.Done := TRUE;
       END_IF;

       // command reset done resets done state and than resets command

       IF #DrainingPhase.Cmd.ResetDone THEN
           #DrainingPhase.State.Done := FALSE;
       END_IF;
       #DrainingPhase.Cmd.ResetDone := FALSE;
   END_REGION

   REGION States 
       //Command valve in cases of states

       IF #DrainingPhase.State.Running THEN
           #DrainingValve.Cmd.Req2OpenAut := TRUE;
           #DrainingValve.Cmd.Req2CloseAut := FALSE;
       ELSE
           #DrainingValve.Cmd.Req2OpenAut := FALSE;
           #DrainingValve.Cmd.Req2CloseAut := TRUE;
       END_IF;
   END_REGION

   // delault state of phase - if not any state sets state to idle

   IF NOT #DrainingPhase.State.Running AND NOT #DrainingPhase.State.Idle AND NOT #DrainingPhase.State.Paused THEN
       #DrainingPhase.State.Idle := TRUE;
   END_IF;

   // write binary states into int value for visualization

   IF #DrainingPhase.State.Running THEN
       #DrainingPhase.State.StateInt := #Running;
   ELSIF #DrainingPhase.State.Idle THEN
       #DrainingPhase.State.StateInt := #Idle;
   ELSE
       #DrainingPhase.State.StateInt := #Pause;
   END_IF;
END_FUNCTION_BLOCK

FUNCTION_BLOCK "MixingFC"   // FB6, SCL
{ S7_Optimized_Access := 'TRUE' }
VERSION : 0.1
   VAR_INPUT
      iSecImp : Bool;
   END_VAR
   VAR_IN_OUT
      MixingPhase : "PhaseMixing";
      MixerEng : "Engine";
   END_VAR
   VAR
      fElapsedTime : Int;
      fSecImp : R_TRIG;
   END_VAR
   VAR CONSTANT
      Idle : Int := 0;
      Running : Int := 1;
      Pause : Int := 2;
   END_VAR
BEGIN
   REGION Aut/Man
       // switching state of engine - automatic or manual control (default state is manual)

       IF (#MixingPhase.Cmd.AutCtrl AND #MixingPhase.Cmd.ManCtrl) OR (NOT #MixingPhase.State.AutCtrl AND NOT #MixingPhase.State.ManCtrl) THEN
           #MixingPhase.State.AutCtrl := FALSE;
           #MixingPhase.State.ManCtrl := TRUE;
       ELSIF #MixingPhase.Cmd.AutCtrl THEN
           #MixingPhase.State.AutCtrl := TRUE;
           #MixingPhase.State.ManCtrl := FALSE;
       ELSIF #MixingPhase.Cmd.ManCtrl THEN
           #MixingPhase.State.AutCtrl := FALSE;
           #MixingPhase.State.ManCtrl := TRUE;
       END_IF;

       #MixingPhase.Cmd.AutCtrl := FALSE;
       #MixingPhase.Cmd.ManCtrl := FALSE;
   END_REGION

   REGION ManCtrl
       // processing manual actions - if command is processed, it is sets to FALSE even if can't be processed
       // Phase commands are start, stop, pause and resume 
       // Start - start mixing  
       // Stop - stop mixing
       // Pause - stop mixing 
       // Resume - start mixing
       // real states of phase are writed into states in phase structure

       IF #MixingPhase.State.ManCtrl THEN
           IF #MixingPhase.Cmd.StartMan AND #MixingPhase.State.Idle THEN
               #MixingPhase.State.Running := TRUE;
               #MixingPhase.State.Idle := FALSE;
               #MixingPhase.State.Paused := FALSE;
               #MixingPhase.State.Done := FALSE;
           ELSIF #MixingPhase.Cmd.StopMan THEN
               #MixingPhase.State.Running := FALSE;
               #MixingPhase.State.Idle := TRUE;
               #MixingPhase.State.Paused := FALSE;
               #MixingPhase.State.Done := FALSE;
               #fElapsedTime := 0;
           ELSIF #MixingPhase.Cmd.PauseMan AND #MixingPhase.State.Running THEN
               #MixingPhase.State.Running := FALSE;
               #MixingPhase.State.Idle := FALSE;
               #MixingPhase.State.Paused := TRUE;
               #MixingPhase.State.Done := FALSE;
           ELSIF #MixingPhase.Cmd.ResumeMan AND #MixingPhase.State.Paused THEN
               #MixingPhase.State.Running := TRUE;
               #MixingPhase.State.Idle := FALSE;
               #MixingPhase.State.Paused := FALSE;
               #MixingPhase.State.Done := FALSE;
           END_IF;
       END_IF;

       #MixingPhase.Cmd.StartMan := FALSE;
       #MixingPhase.Cmd.StopMan := FALSE;
       #MixingPhase.Cmd.PauseMan := FALSE;
       #MixingPhase.Cmd.ResumeMan := FALSE;
   END_REGION

   REGION AutCtrl
       // if request to run in automatic mode -> set auto request to mixing to 1, if not request to mixing is 0
       // commands should be sets to false after their processing

       IF #MixingPhase.State.AutCtrl THEN
           IF #MixingPhase.Cmd.StartAut THEN
               #MixingPhase.State.Running := TRUE;
               #MixingPhase.State.Idle := FALSE;
               #MixingPhase.State.Paused := FALSE;
               #MixingPhase.State.Done := FALSE;
           ELSIF #MixingPhase.Cmd.StopAut THEN
               #MixingPhase.State.Running := FALSE;
               #MixingPhase.State.Idle := TRUE;
               #MixingPhase.State.Paused := FALSE;
               #MixingPhase.State.Done := FALSE;
               #fElapsedTime := 0;
           END_IF;
       END_IF;

       #MixingPhase.Cmd.StartAut := FALSE;
       #MixingPhase.Cmd.StopAut := FALSE;
   END_REGION


   REGION Done
       // every phase should have finish condition - mixing phase - if time of runnig is bigger or same as requested
       // after that done state should be setted to 1

       #fSecImp(CLK := #iSecImp);
       IF #fSecImp.Q AND #MixingPhase.State.Running AND NOT (#MixingPhase.Param.TimeSec = -1) THEN
           #fElapsedTime += 1;
       END_IF;

       IF #MixingPhase.State.Running AND #fElapsedTime >= #MixingPhase.Param.TimeSec AND NOT (#MixingPhase.Param.TimeSec = -1) THEN
           #MixingPhase.Cmd.StopAut := TRUE;
           #MixingPhase.Cmd.StopMan := TRUE;
           #MixingPhase.State.Done := TRUE;
       END_IF;

       IF #MixingPhase.State.Paused OR #MixingPhase.State.Idle THEN
           #MixingPhase.State.Done := TRUE;
       END_IF;

       // command reset done resets done state and than resets command

       IF #MixingPhase.Cmd.ResetDone THEN
           #MixingPhase.State.Done := FALSE;
       END_IF;
       #MixingPhase.Cmd.ResetDone := FALSE;
   END_REGION

   REGION States 
       //Command mixer in cases of states

       IF #MixingPhase.State.Running THEN
           #MixerEng.Cmd.Req2RunAutCtrl := TRUE;
       ELSE
           #MixerEng.Cmd.Req2RunAutCtrl := FALSE;
       END_IF;
   END_REGION

   // delault state of phase - if not any state sets state to idle

   IF NOT #MixingPhase.State.Running AND NOT #MixingPhase.State.Idle AND NOT #MixingPhase.State.Paused THEN
       #MixingPhase.State.Idle := TRUE;
   END_IF;

   // write binary states into int value for visualization

   IF #MixingPhase.State.Running THEN
       #MixingPhase.State.StateInt := #Running;
   ELSIF #MixingPhase.State.Idle THEN
       #MixingPhase.State.StateInt := #Idle;
   ELSE
       #MixingPhase.State.StateInt := #Pause;
   END_IF;
END_FUNCTION_BLOCK

FUNCTION_BLOCK "HeaterFC"   // FB7, SCL
{ S7_Optimized_Access := 'TRUE' }
VERSION : 0.1
   VAR_INPUT
      iWaterTemp : Real;
   END_VAR
   VAR_OUTPUT
      oHeaterEnable : Bool;
      oHeaterPower : Real;
   END_VAR
   VAR_IN_OUT
      iHeater_Struct : "Heater";
   END_VAR
   VAR
      fMode : Int;
   END_VAR
BEGIN
   #fMode := 3; // automatic mode of PID component
   "HeatingPID"(Setpoint := #iHeater_Struct.Param.HeatingSetPointAutomat,
                Input := #iWaterTemp,
                ManualEnable := #iHeater_Struct.State.ManCtrl,
                ManualValue := #iHeater_Struct.Param.HeatingPowerManual,
                OutputHeat => #iHeater_Struct.State.HeatingOut,
                Mode := #fMode);

   REGION Manual/Automat

       IF (#iHeater_Struct.Cmd.AutCtrl AND #iHeater_Struct.Cmd.ManCtrl) OR (NOT #iHeater_Struct.State.AutCtrl AND NOT #iHeater_Struct.State.ManCtrl) THEN
           #iHeater_Struct.State.AutCtrl := FALSE;
           #iHeater_Struct.State.ManCtrl := TRUE;
       ELSIF #iHeater_Struct.Cmd.AutCtrl THEN
           #iHeater_Struct.State.AutCtrl := TRUE;
           #iHeater_Struct.State.ManCtrl := FALSE;
       ELSIF #iHeater_Struct.Cmd.ManCtrl THEN
           #iHeater_Struct.State.AutCtrl := FALSE;
           #iHeater_Struct.State.ManCtrl := TRUE;
       END_IF;

       #iHeater_Struct.Cmd.AutCtrl := FALSE;
       #iHeater_Struct.Cmd.ManCtrl := FALSE;
   END_REGION

   REGION ManCtrl

       IF #iHeater_Struct.Cmd.TurnOnMan AND #iHeater_Struct.State.ManCtrl THEN
           // set the state
           #iHeater_Struct.State.EnableOut := TRUE;
       END_IF;

       IF #iHeater_Struct.Cmd.TurnOffMan AND #iHeater_Struct.State.ManCtrl THEN
           #iHeater_Struct.State.EnableOut := FALSE;
       END_IF;

       #iHeater_Struct.Cmd.TurnOnMan := FALSE;
       #iHeater_Struct.Cmd.TurnOffMan := FALSE;
   END_REGION

   REGION AutCtrl

       IF #iHeater_Struct.State.AutCtrl THEN
           #iHeater_Struct.State.EnableOut := #iHeater_Struct.Cmd.Req2RunAutCtrl;
       END_IF;
   END_REGION

   #oHeaterEnable := #iHeater_Struct.State.EnableOut;
   #oHeaterPower := #iHeater_Struct.State.HeatingOut;
END_FUNCTION_BLOCK

FUNCTION_BLOCK "Real2AnalogValue"   // FB8, SCL
{ S7_Optimized_Access := 'TRUE' }
VERSION : 0.1
   VAR_INPUT
      aiRealValue : Real;
      TransducerLoLevel : Int;
      TransducerHiLevel : Int;
      ScaledValLoLevel : Real;
      ScaledValHiLevel : Real;
   END_VAR
   VAR_OUTPUT
      aoRawAnalog : Int;
   END_VAR
BEGIN
   #aoRawAnalog := REAL_TO_INT(((#TransducerHiLevel - #TransducerLoLevel) / (#ScaledValHiLevel - #ScaledValLoLevel)) * (#aiRealValue - #ScaledValLoLevel) + #TransducerLoLevel);
END_FUNCTION_BLOCK

FUNCTION_BLOCK "HeatingFC"   // FB9, SCL
{ S7_Optimized_Access := 'TRUE' }
VERSION : 0.1
   VAR_INPUT
      iSecImp : Bool;
      aiWaterTemp : Real;
   END_VAR
   VAR_IN_OUT
      HeatingPhase : "PhaseHeating";
      Heater : "Heater";
   END_VAR
   VAR
      fTime : Int;
      fSecImpEdge : R_TRIG;
   END_VAR
   VAR CONSTANT
      Idle : Int := 0;
      Running : Int := 1;
      Pause : Int := 2;
   END_VAR
BEGIN
   REGION Aut/Man
       // switching state of engine - automatic or manual control (default state is manual)

       IF (#HeatingPhase.Cmd.AutCtrl AND #HeatingPhase.Cmd.ManCtrl) OR (NOT #HeatingPhase.State.AutCtrl AND NOT #HeatingPhase.State.ManCtrl) THEN
           #HeatingPhase.State.AutCtrl := FALSE;
           #HeatingPhase.State.ManCtrl := TRUE;
       ELSIF #HeatingPhase.Cmd.AutCtrl THEN
           #HeatingPhase.State.AutCtrl := TRUE;
           #HeatingPhase.State.ManCtrl := FALSE;
       ELSIF #HeatingPhase.Cmd.ManCtrl THEN
           #HeatingPhase.State.AutCtrl := FALSE;
           #HeatingPhase.State.ManCtrl := TRUE;
       END_IF;

       #HeatingPhase.Cmd.AutCtrl := FALSE;
       #HeatingPhase.Cmd.ManCtrl := FALSE;
   END_REGION

   REGION ManCtrl
       // processing manual actions - if command is processed, it is sets to FALSE even if can't be processed
       // real states of phase are writed into states in phase structure

       IF #HeatingPhase.State.ManCtrl THEN
           IF #HeatingPhase.Cmd.StartMan AND #HeatingPhase.State.Idle THEN
               #HeatingPhase.State.Running := TRUE;
               #HeatingPhase.State.Idle := FALSE;
               #HeatingPhase.State.Paused := FALSE;
               #HeatingPhase.State.Done := FALSE;
           ELSIF #HeatingPhase.Cmd.StopMan THEN
               #HeatingPhase.State.Running := FALSE;
               #HeatingPhase.State.Idle := TRUE;
               #HeatingPhase.State.Paused := FALSE;
               #HeatingPhase.State.Done := FALSE;
           ELSIF #HeatingPhase.Cmd.PauseMan AND #HeatingPhase.State.Running THEN
               #HeatingPhase.State.Running := FALSE;
               #HeatingPhase.State.Idle := FALSE;
               #HeatingPhase.State.Paused := TRUE;
               #HeatingPhase.State.Done := FALSE;
           ELSIF #HeatingPhase.Cmd.ResumeMan AND #HeatingPhase.State.Paused THEN
               #HeatingPhase.State.Running := TRUE;
               #HeatingPhase.State.Idle := FALSE;
               #HeatingPhase.State.Paused := FALSE;
               #HeatingPhase.State.Done := FALSE;
           END_IF;
       END_IF;

       #HeatingPhase.Cmd.StartMan := FALSE;
       #HeatingPhase.Cmd.StopMan := FALSE;
       #HeatingPhase.Cmd.PauseMan := FALSE;
       #HeatingPhase.Cmd.ResumeMan := FALSE;
   END_REGION

   REGION AutCtrl
       // if request to run in automatic mode -> set auto request to heat to 1, if not request to heat 0
       // commands should be sets to false after their processing

       IF #HeatingPhase.State.AutCtrl THEN
           IF #HeatingPhase.Cmd.StartAut THEN
               #HeatingPhase.State.Running := TRUE;
               #HeatingPhase.State.Idle := FALSE;
               #HeatingPhase.State.Paused := FALSE;
               #HeatingPhase.State.Done := FALSE;
           ELSIF #HeatingPhase.Cmd.StopAut THEN
               #HeatingPhase.State.Running := FALSE;
               #HeatingPhase.State.Idle := TRUE;
               #HeatingPhase.State.Paused := FALSE;
               #HeatingPhase.State.Done := FALSE;
           END_IF;
       END_IF;

       #HeatingPhase.Cmd.StartAut := FALSE;
       #HeatingPhase.Cmd.StopAut := FALSE;
   END_REGION

   REGION Done
       //every phase should have finish condition - heating phase - if water temp is on requested value for 10 seconds with 1°C hysteresis
       //after that done state should be setted to 1

       #fSecImpEdge(CLK := #iSecImp);
       IF #fSecImpEdge.Q AND #HeatingPhase.State.Running THEN
           #fTime += 1;
       END_IF;

       IF ABS(#aiWaterTemp - #Heater.Param.HeatingSetPointAutomat) > 1.0 OR NOT #HeatingPhase.State.Running THEN
           #fTime := 0;
       END_IF;

       IF #fTime >= 10 AND #HeatingPhase.State.Running THEN
           #HeatingPhase.State.Done := TRUE;
       END_IF;

       IF #HeatingPhase.State.Paused OR #HeatingPhase.State.Idle THEN
           #HeatingPhase.State.Done := TRUE;
       END_IF;

       // command reset done resets done state and than resets command

       IF #HeatingPhase.Cmd.ResetDone THEN
           #HeatingPhase.State.Done := FALSE;
           #fTime := 0;
       END_IF;
       #HeatingPhase.Cmd.ResetDone := FALSE;
   END_REGION

   REGION States 
       //Command valve in cases of states
       // Running - start heating  
       // Idle - stop heating
       // Pause - stop heating (alternative is hold actual temp)

       IF #HeatingPhase.State.Running THEN
           #Heater.Cmd.Req2RunAutCtrl := TRUE;
       ELSE
           #Heater.Cmd.Req2RunAutCtrl := FALSE;
       END_IF;
   END_REGION

   // delault state of phase - if not any state sets state to idle

   IF NOT #HeatingPhase.State.Running AND NOT #HeatingPhase.State.Idle AND NOT #HeatingPhase.State.Paused THEN
       #HeatingPhase.State.Idle := TRUE;
   END_IF;

   // write binary states into int value for visualization

   IF #HeatingPhase.State.Running THEN
       #HeatingPhase.State.StateInt := #Running;
   ELSIF #HeatingPhase.State.Idle THEN
       #HeatingPhase.State.StateInt := #Idle;
   ELSE
       #HeatingPhase.State.StateInt := #Pause;
   END_IF;
END_FUNCTION_BLOCK

FUNCTION "AnalogScalingFC" : Void   // FC1, SCL
{ S7_Optimized_Access := 'TRUE' }
VERSION : 0.1
   VAR_INPUT
      aiRAWanalog : Int;
      TransducerLoLevel : Int;
      TransducerHiLevel : Int;
      ScaledValLoLevel : Real;
      ScaledValHiLevel : Real;
   END_VAR
   VAR_OUTPUT
      aoScaledValue : Real;
   END_VAR
BEGIN
   #aoScaledValue := ((#ScaledValHiLevel-#ScaledValLoLevel)/(#TransducerHiLevel-#TransducerLoLevel))*(#aiRAWanalog-#TransducerLoLevel)+#ScaledValLoLevel;
END_FUNCTION

(* ===== HMI "HMI_RT_1" =====
system functions are stored by id; their names below are inferred from use
connection "HMI_Connection_2": ETHERNET, S7_1500_OMS

HMI tags "Default tag table"
   "Tag_ScreenNumber" : UInt, internal
   "Data_Tank1_ValveFill_State_AutCtrl" : Bool = PLC Data.Tank1.ValveFill.State.AutCtrl, 100 ms
   "Data_Tank1_ValveFill_State_ManCtrl" : Bool = PLC Data.Tank1.ValveFill.State.ManCtrl, 100 ms
   "Data_Tank1_ValveFill_State_Open" : Bool = PLC Data.Tank1.ValveFill.State.Open, 100 ms
   "Data_Tank1_ValveFill_State_Closed" : Bool = PLC Data.Tank1.ValveFill.State.Closed, 100 ms
   "Data_Tank1_Mixer_State_AutCtrl" : Bool = PLC Data.Tank1.Mixer.State.AutCtrl, 100 ms
   "Data_Tank1_Mixer_State_ManCtrl" : Bool = PLC Data.Tank1.Mixer.State.ManCtrl, 100 ms
   "Data_Tank1_Mixer_State_Run" : Bool = PLC Data.Tank1.Mixer.State.Run, 100 ms
   "Data_Tank1_ValveDrain_State_AutCtrl" : Bool = PLC Data.Tank1.ValveDrain.State.AutCtrl, 100 ms
   "Data_Tank1_ValveDrain_State_ManCtrl" : Bool = PLC Data.Tank1.ValveDrain.State.ManCtrl, 100 ms
   "Data_Tank1_ValveDrain_State_Open" : Bool = PLC Data.Tank1.ValveDrain.State.Open, 100 ms
   "Data_Tank1_ValveDrain_State_Closed" : Bool = PLC Data.Tank1.ValveDrain.State.Closed, 100 ms
   "Data_Tank1_ValveFill_Cmd_AutCtrl" : Bool = PLC Data.Tank1.ValveFill.Cmd.AutCtrl, 100 ms
   "Data_Tank1_ValveFill_Cmd_ManCtrl" : Bool = PLC Data.Tank1.ValveFill.Cmd.ManCtrl, 100 ms
   "Data_Tank1_ValveFill_Cmd_OpenMan" : Bool = PLC Data.Tank1.ValveFill.Cmd.OpenMan, 100 ms
   "Data_Tank1_ValveFill_Cmd_CloseMan" : Bool = PLC Data.Tank1.ValveFill.Cmd.CloseMan, 100 ms
   "Data_Tank1_Mixer_Cmd_AutCtrl" : Bool = PLC Data.Tank1.Mixer.Cmd.AutCtrl, 100 ms
   "Data_Tank1_Mixer_Cmd_ManCtrl" : Bool = PLC Data.Tank1.Mixer.Cmd.ManCtrl, 100 ms
   "Data_Tank1_Mixer_Cmd_TurnOnMan" : Bool = PLC Data.Tank1.Mixer.Cmd.TurnOnMan, 100 ms
   "Data_Tank1_Mixer_Cmd_TurnOffMan" : Bool = PLC Data.Tank1.Mixer.Cmd.TurnOffMan, 100 ms
   "Data_Tank1_ValveDrain_Cmd_AutCtrl" : Bool = PLC Data.Tank1.ValveDrain.Cmd.AutCtrl, 100 ms
   "Data_Tank1_ValveDrain_Cmd_OpenMan" : Bool = PLC Data.Tank1.ValveDrain.Cmd.OpenMan, 100 ms
   "Data_Tank1_ValveDrain_Cmd_CloseMan" : Bool = PLC Data.Tank1.ValveDrain.Cmd.CloseMan, 100 ms
   "Data_Tank1_WaterLevel_AIScaled" : Real = PLC Data.Tank1.WaterLevel.AIScaled, 100 ms
   "Data_Tank1_WaterTemp_AIScaled" : Real = PLC Data.Tank1.WaterTemp.AIScaled, 100 ms
   "HeatingPID_ManualEnable" : Bool = PLC HeatingPID.ManualEnable, 100 ms
   "Data_Tank1_Heating_Param_ReqTemp" : Real = PLC Data.Tank1.Heating.Param.ReqTemp, 100 ms
   "Data_Tank1_Filling_State_Stateint" : Int = PLC Data.Tank1.Filling.State.Stateint, 100 ms
   "Data_Tank1_Draining_State_StateInt" : Int = PLC Data.Tank1.Draining.State.StateInt, 100 ms
   "Data_Tank1_Mixing_State_StateInt" : Int = PLC Data.Tank1.Mixing.State.StateInt, 100 ms
   "Data_Tank1_Heating_State_StateInt" : Int = PLC Data.Tank1.Heating.State.StateInt, 100 ms
   "Data_Tank1_Filling_State_AutCtrl" : Bool = PLC Data.Tank1.Filling.State.AutCtrl, 100 ms
   "Data_Tank1_Filling_State_ManCtrl" : Bool = PLC Data.Tank1.Filling.State.ManCtrl, 100 ms
   "Data_Tank1_Filling_State_Done" : Bool = PLC Data.Tank1.Filling.State.Done, 100 ms
   "Data_Tank1_Filling_Cmd_AutCtrl" : Bool = PLC Data.Tank1.Filling.Cmd.AutCtrl, 100 ms
   "Data_Tank1_Filling_Cmd_ManCtrl" : Bool = PLC Data.Tank1.Filling.Cmd.ManCtrl, 100 ms
   "Data_Tank1_Filling_Cmd_ResetDone" : Bool = PLC Data.Tank1.Filling.Cmd.ResetDone, 100 ms
   "Data_Tank1_Filling_Cmd_StartMan" : Bool = PLC Data.Tank1.Filling.Cmd.StartMan, 100 ms
   "Data_Tank1_Filling_Cmd_StopMan" : Bool = PLC Data.Tank1.Filling.Cmd.StopMan, 100 ms
   "Data_Tank1_Filling_Cmd_PauseMan" : Bool = PLC Data.Tank1.Filling.Cmd.PauseMan, 100 ms
   "Data_Tank1_Filling_Cmd_ResumeMan" : Bool = PLC Data.Tank1.Filling.Cmd.ResumeMan, 100 ms
   "Data_Tank1_Mixing_State_AutCtrl" : Bool = PLC Data.Tank1.Mixing.State.AutCtrl, 100 ms
   "Data_Tank1_Mixing_State_ManCtrl" : Bool = PLC Data.Tank1.Mixing.State.ManCtrl, 100 ms
   "Data_Tank1_Mixing_State_Done" : Bool = PLC Data.Tank1.Mixing.State.Done, 100 ms
   "Data_Tank1_Mixing_Cmd_AutCtrl" : Bool = PLC Data.Tank1.Mixing.Cmd.AutCtrl, 100 ms
   "Data_Tank1_Mixing_Cmd_ManCtrl" : Bool = PLC Data.Tank1.Mixing.Cmd.ManCtrl, 100 ms
   "Data_Tank1_Mixing_Cmd_ResetDone" : Bool = PLC Data.Tank1.Mixing.Cmd.ResetDone, 100 ms
   "Data_Tank1_Mixing_Cmd_StartMan" : Bool = PLC Data.Tank1.Mixing.Cmd.StartMan, 100 ms
   "Data_Tank1_Mixing_Cmd_StopMan" : Bool = PLC Data.Tank1.Mixing.Cmd.StopMan, 100 ms
   "Data_Tank1_Mixing_Cmd_PauseMan" : Bool = PLC Data.Tank1.Mixing.Cmd.PauseMan, 100 ms
   "Data_Tank1_Mixing_Cmd_ResumeMan" : Bool = PLC Data.Tank1.Mixing.Cmd.ResumeMan, 100 ms
   "Data_Tank1_Draining_State_AutCtrl" : Bool = PLC Data.Tank1.Draining.State.AutCtrl, 100 ms
   "Data_Tank1_Draining_State_ManCtrl" : Bool = PLC Data.Tank1.Draining.State.ManCtrl, 100 ms
   "Data_Tank1_Draining_State_Done" : Bool = PLC Data.Tank1.Draining.State.Done, 100 ms
   "Data_Tank1_Draining_Cmd_AutCtrl" : Bool = PLC Data.Tank1.Draining.Cmd.AutCtrl, 100 ms
   "Data_Tank1_Draining_Cmd_ManCtrl" : Bool = PLC Data.Tank1.Draining.Cmd.ManCtrl, 100 ms
   "Data_Tank1_Draining_Cmd_ResetDone" : Bool = PLC Data.Tank1.Draining.Cmd.ResetDone, 100 ms
   "Data_Tank1_Draining_Cmd_StartMan" : Bool = PLC Data.Tank1.Draining.Cmd.StartMan, 100 ms
   "Data_Tank1_Draining_Cmd_StopMan" : Bool = PLC Data.Tank1.Draining.Cmd.StopMan, 100 ms
   "Data_Tank1_Draining_Cmd_PauseMan" : Bool = PLC Data.Tank1.Draining.Cmd.PauseMan, 100 ms
   "Data_Tank1_Draining_Cmd_ResumeMan" : Bool = PLC Data.Tank1.Draining.Cmd.ResumeMan, 100 ms
   "Data_Tank1_Heating_State_AutCtrl" : Bool = PLC Data.Tank1.Heating.State.AutCtrl, 100 ms
   "Data_Tank1_Heating_State_ManCtrl" : Bool = PLC Data.Tank1.Heating.State.ManCtrl, 100 ms
   "Data_Tank1_Heating_State_Done" : Bool = PLC Data.Tank1.Heating.State.Done, 100 ms
   "Data_Tank1_Heating_Cmd_AutCtrl" : Bool = PLC Data.Tank1.Heating.Cmd.AutCtrl, 100 ms
   "Data_Tank1_Heating_Cmd_ManCtrl" : Bool = PLC Data.Tank1.Heating.Cmd.ManCtrl, 100 ms
   "Data_Tank1_Heating_Cmd_ResetDone" : Bool = PLC Data.Tank1.Heating.Cmd.ResetDone, 100 ms
   "Data_Tank1_Heating_Cmd_StartMan" : Bool = PLC Data.Tank1.Heating.Cmd.StartMan, 100 ms
   "Data_Tank1_Heating_Cmd_StopMan" : Bool = PLC Data.Tank1.Heating.Cmd.StopMan, 100 ms
   "Data_Tank1_Heating_Cmd_PauseMan" : Bool = PLC Data.Tank1.Heating.Cmd.PauseMan, 100 ms
   "Data_Tank1_Heating_Cmd_ResumeMan" : Bool = PLC Data.Tank1.Heating.Cmd.ResumeMan, 100 ms
   "Data_Tank1_Filling_Param_FillLevel" : Real = PLC Data.Tank1.Filling.Param.FillLevel, 100 ms
   "Data_Tank1_Draining_Param_DrainLevel" : Real = PLC Data.Tank1.Draining.Param.DrainLevel, 100 ms
   "Data_Tank1_Mixing_Param_TimeSec" : Int = PLC Data.Tank1.Mixing.Param.TimeSec, 100 ms
   "Data_Tank1_Mixer_State_StateInt" : Int = PLC Data.Tank1.Mixer.State.StateInt, 100 ms
   "Data_Tank1_ValveFill_State_StColor" : Int = PLC Data.Tank1.ValveFill.State.StColor, 100 ms
   "Data_Tank1_ValveDrain_State_StColor" : Int = PLC Data.Tank1.ValveDrain.State.StColor, 100 ms
   "Data_Tank1_ValveDrain_Cmd_ManCtrl" : Bool = PLC Data.Tank1.ValveDrain.Cmd.ManCtrl, 100 ms
   "Data_Tank1_Heater_Cmd_AutCtrl" : Bool = PLC Data.Tank1.Heater.Cmd.AutCtrl, 100 ms
   "Data_Tank1_Heater_Cmd_ManCtrl" : Bool = PLC Data.Tank1.Heater.Cmd.ManCtrl, 100 ms
   "Data_Tank1_Heater_Cmd_TurnOnMan" : Bool = PLC Data.Tank1.Heater.Cmd.TurnOnMan, 100 ms
   "Data_Tank1_Heater_Cmd_TurnOffMan" : Bool = PLC Data.Tank1.Heater.Cmd.TurnOffMan, 100 ms
   "Data_Tank1_Heater_Param_HeatingPowerManual" : Real = PLC Data.Tank1.Heater.Param.HeatingPowerManual, 100 ms
   "Data_Tank1_Heater_State_AutCtrl" : Bool = PLC Data.Tank1.Heater.State.AutCtrl, 100 ms
   "Data_Tank1_Heater_State_ManCtrl" : Bool = PLC Data.Tank1.Heater.State.ManCtrl, 100 ms
   "Data_ProcessControl1_Cmd_Start" : Bool = PLC Data.ProcessControl1.Cmd.Start AT %DB1.DBW0, 100 ms
   "Data_ProcessControl1_Cmd_Stop" : Bool = PLC Data.ProcessControl1.Cmd.Stop AT %DB1.DBX0.0, 1 s
   "Data_ProcessControl1_State_Phase" : Int = PLC Data.ProcessControl1.State.Phase AT %DB1.DBX0.0, 1 s
   "Data_Tank1_Heater_Param_HeatingSetPointAutomat" : Real = PLC Data.Tank1.Heater.Param.HeatingSetPointAutomat AT %DB1.DBD0, 1 s

text list "Phases": 0 'Idle'; 1 'Running'; 2 'Pause'

text list "Process": 0 'Running'; 1 'Idle'; 2 'Stopping'

text list "Phases_Control": 0 'Idle'; 1..10 'Running'

screen "MainScr" 800x480
   SymbolLibrary "Symbol library_1" at 202,63 size 120x212
   SymbolLibrary "Symbol library_2" at 148,84 size 58x23
   SymbolLibrary "Symbol library_3" at 320,241 size 25x23
   Bar "Bar_1" at 204,63 size 117x211; MinimumValue 0; MaximumValue 2
      ProcessValue <- "Data_Tank1_WaterLevel_AIScaled"
   SymbolLibrary "Symbol library_4" at 55,31 size 94x80
      Appearance <- "Data_Tank1_ValveFill_State_StColor"
   IOField "I/O field_1" at 215,109 size 96x32; FormatPattern s9.99; Unit  m
      ProcessValue <- "Data_Tank1_WaterLevel_AIScaled"
   IOField "I/O field_2" at 216,143 size 96x32; FormatPattern 999.9; Unit  °C
      ProcessValue <- "Data_Tank1_WaterTemp_AIScaled"
   SymbolLibrary "Symbol library_6" at 226,190 size 71x61
      Appearance <- "Data_Tank1_Mixer_State_StateInt"
   Button "Button_1" at 7,233 size 77x32; TextOff 'Aut'
      on Click: SetBit("Data_Tank1_ValveFill_Cmd_AutCtrl")
   TextField "Text field_1" at 45,123 size 83x23; Text 'ValveFill'
   TextField "Text field_2" at 5,148 size 83x23; Text 'Automat'
   TextField "Text field_3" at 5,166 size 70x23; Text 'Manual'
   TextField "Text field_4" at 5,188 size 51x23; Text 'Open'
   TextField "Text field_5" at 5,206 size 65x23; Text 'Closed'
   Button "Button_2" at 86,233 size 77x32; TextOff 'Man'
      on Click: SetBit("Data_Tank1_ValveFill_Cmd_ManCtrl")
   Button "Button_3" at 7,267 size 77x32; TextOff 'Open'
      on Click: SetBit("Data_Tank1_ValveFill_Cmd_OpenMan")
   Button "Button_4" at 86,267 size 77x32; TextOff 'Close'
      on Click: SetBit("Data_Tank1_ValveFill_Cmd_CloseMan")
   Circle "Circle_1" at 122,149 size 20x20
      Appearance <- "Data_Tank1_ValveFill_State_AutCtrl"
   Circle "Circle_2" at 122,169 size 20x20
      Appearance <- "Data_Tank1_ValveFill_State_ManCtrl"
   Circle "Circle_3" at 122,189 size 20x20
      Appearance <- "Data_Tank1_ValveFill_State_Open"
   Circle "Circle_4" at 122,209 size 20x20
      Appearance <- "Data_Tank1_ValveFill_State_Closed"
   TextField "Text field_6" at 450,99 size 104x23; Text 'ValveDrain'
   TextField "Text field_7" at 417,124 size 83x23; Text 'Automat'
   TextField "Text field_8" at 417,142 size 70x23; Text 'Manual'
   TextField "Text field_9" at 417,164 size 51x23; Text 'Open'
   TextField "Text field_10" at 417,182 size 65x23; Text 'Closed'
   TextField "Text field_11" at 234,284 size 56x23; Text 'Mixer'
   TextField "Text field_12" at 185,309 size 83x23; Text 'Automat'
   TextField "Text field_13" at 185,327 size 70x23; Text 'Manual'
   TextField "Text field_14" at 185,350 size 79x23; Text 'Running'
   Circle "Circle_9" at 302,310 size 20x20
      Appearance <- "Data_Tank1_Mixer_State_AutCtrl"
   Circle "Circle_10" at 302,330 size 20x20
      Appearance <- "Data_Tank1_Mixer_State_ManCtrl"
   Circle "Circle_12" at 302,354 size 20x20
      Appearance <- "Data_Tank1_Mixer_State_Run"
   TextField "Text field_16" at 626,95 size 77x27; Text 'Phases'
   Button "Button_15" at 617,148 size 128x29; TextOff 'Menu'
      on Click: ActivateScreen("Filling", 0)
   TextField "Text field_17" at 655,124 size 61x23; Text 'Filling'
   SymbolicIOField "Symbolic I/O field_2" at 617,179 size 129x32; TextOn '1'; TextOff '0'; TextList "Phases"
      ProcessValue <- "Data_Tank1_Filling_State_Stateint"
   Button "Button_16" at 617,236 size 129x29; TextOff 'Menu'
      on Click: ActivateScreen("Draining", 0)
   TextField "Text field_18" at 642,213 size 82x23; Text 'Draining'
   SymbolicIOField "Symbolic I/O field_3" at 617,267 size 129x32; TextOn '1'; TextOff '0'; TextList "Phases"
      ProcessValue <- "Data_Tank1_Draining_State_StateInt"
   Button "Button_17" at 617,324 size 130x29; TextOff 'Menu'
      on Click: ActivateScreen("Mixing", 0)
   TextField "Text field_19" at 650,302 size 65x23; Text 'Mixing'
   SymbolicIOField "Symbolic I/O field_4" at 617,355 size 130x32; TextOn '1'; TextOff '0'; TextList "Phases"
      ProcessValue <- "Data_Tank1_Mixing_State_StateInt"
   TextField "Text field_21" at 427,285 size 156x23; Text 'Heating element'
   TextField "Text field_22" at 418,310 size 83x23; Text 'Automat'
   TextField "Text field_23" at 418,328 size 70x23; Text 'Manual'
   TextField "Text field_24" at 422,350 size 157x23; Text 'Manual heat pwr'
   IOField "I/O field_3" at 447,371 size 96x32; FormatPattern 999; Unit  %
      ProcessValue <- "Data_Tank1_Heater_Param_HeatingPowerManual"
   Button "Button_19" at 435,16 size 130x66; TextOff 'Parameters tank 1'
      on Click: ActivateScreen("Parameters", 0)
   SymbolLibrary "Symbol library_5" at 319,188 size 94x80
      Appearance <- "Data_Tank1_ValveDrain_State_StColor"
   SymbolLibrary "Symbol library_7" at 23,84 size 58x23
   Circle "Circle_5" at 543,125 size 20x20
      Appearance <- "Data_Tank1_ValveDrain_State_AutCtrl"
   Circle "Circle_6" at 543,145 size 20x20
      Appearance <- "Data_Tank1_ValveDrain_State_ManCtrl"
   Circle "Circle_7" at 543,165 size 20x20
      Appearance <- "Data_Tank1_ValveDrain_State_Open"
   Circle "Circle_8" at 543,185 size 20x20
      Appearance <- "Data_Tank1_ValveDrain_State_Closed"
   Button "Button_5" at 187,377 size 77x32; TextOff 'Aut'
      on Click: SetBit("Data_Tank1_Mixer_Cmd_AutCtrl")
   Button "Button_6" at 266,377 size 77x32; TextOff 'Man'
      on Click: SetBit("Data_Tank1_Mixer_Cmd_ManCtrl")
   Button "Button_7" at 187,411 size 77x32; TextOff 'On'
      on Click: SetBit("Data_Tank1_Mixer_Cmd_TurnOnMan")
   Button "Button_8" at 266,411 size 77x32; TextOff 'Off'
      on Click: SetBit("Data_Tank1_Mixer_Cmd_TurnOffMan")
   Button "Button_9" at 420,210 size 77x32; TextOff 'Aut'
      on Click: SetBit("Data_Tank1_ValveDrain_Cmd_AutCtrl")
   Button "Button_10" at 499,210 size 77x32; TextOff 'Man'
      on Click: SetBit("Data_Tank1_ValveDrain_Cmd_ManCtrl")
   Button "Button_11" at 420,244 size 77x32; TextOff 'Open'
      on Click: SetBit("Data_Tank1_ValveDrain_Cmd_OpenMan")
   Button "Button_12" at 499,244 size 77x32; TextOff 'Close'
      on Click: SetBit("Data_Tank1_ValveDrain_Cmd_CloseMan")
   Circle "Circle_11" at 542,312 size 20x20
      Appearance <- "Data_Tank1_Heater_State_AutCtrl"
   Circle "Circle_13" at 542,332 size 20x20
      Appearance <- "Data_Tank1_Heater_State_ManCtrl"
   Button "Button_13" at 420,407 size 77x32; TextOff 'Aut'
      on Click: SetBit("Data_Tank1_Heater_Cmd_AutCtrl")
   Button "Button_14" at 499,407 size 77x32; TextOff 'Man'
      on Click: SetBit("Data_Tank1_Heater_Cmd_ManCtrl")
   Button "Button_20" at 420,441 size 77x32; TextOff 'On'
      on Click: SetBit("Data_Tank1_Heater_Cmd_TurnOnMan")
   Button "Button_21" at 499,441 size 77x32; TextOff 'Off'
      on Click: SetBit("Data_Tank1_Heater_Cmd_TurnOffMan")
   Button "Button_18" at 617,412 size 130x29; TextOff 'Menu'
      on Click: ActivateScreen("Heating", 0)
   SymbolicIOField "Symbolic I/O field_5" at 617,443 size 130x32; TextOn '1'; TextOff '0'; TextList "Phases"
      ProcessValue <- "Data_Tank1_Heating_State_StateInt"
   TextField "Text field_20" at 647,390 size 76x23; Text 'Heating'
   Circle "Circle_14" at 761,167 size 20x20
      Appearance <- "Data_Tank1_Filling_State_Done"
   TextField "Text field_15" at 734,95 size 58x27; Text 'Done'
   Circle "Circle_15" at 762,258 size 20x20
      Appearance <- "Data_Tank1_Draining_State_Done"
   Circle "Circle_16" at 761,344 size 20x20
      Appearance <- "Data_Tank1_Mixing_State_Done"
   Circle "Circle_17" at 762,433 size 20x20
      Appearance <- "Data_Tank1_Heating_State_Done"
   Button "Button_22" at 624,16 size 74x29; TextOff 'Start'
      on Click: SetBit("Data_ProcessControl1_Cmd_Start")
   Button "Button_23" at 706,16 size 74x29; TextOff 'Stop'
      on Click: SetBit("Data_ProcessControl1_Cmd_Stop")
   SymbolicIOField "Symbolic I/O field_1" at 642,50 size 129x32; TextOn '1'; TextOff '0'; TextList "Phases_Control"
      ProcessValue <- "Data_ProcessControl1_State_Phase"

screen "Heating" 800x480
   TextField "Text field_26" at 212,181 size 205x23; Text 'Heating phase control'
   TextField "Text field_27" at 116,215 size 83x23; Text 'Automat'
   TextField "Text field_28" at 116,233 size 70x23; Text 'Manual'
   TextField "Text field_29" at 277,224 size 51x23; Text 'Done'
   GraphicView "Graphic view_1" at 459,176 size 75x74; Picture "exit-png-cancel-cross-exit-remove-icon-512"
   Button "Button_19" at 117,262 size 77x32; TextOff 'Aut'
      on Click: SetBit("Data_Tank1_Heating_Cmd_AutCtrl")
   Button "Button_20" at 197,262 size 77x32; TextOff 'Man'
      on Click: SetBit("Data_Tank1_Heating_Cmd_ManCtrl")
   Circle "Circle_14" at 233,216 size 20x20
      Appearance <- "Data_Tank1_Heating_State_AutCtrl"
   Circle "Circle_15" at 233,236 size 20x20
      Appearance <- "Data_Tank1_Heating_State_ManCtrl"
   Button "Button_21" at 278,262 size 157x32; TextOff 'Reset done'
      on Click: SetBit("Data_Tank1_Heating_Cmd_ResetDone")
   Button "Button_22" at 117,312 size 77x32; TextOff 'Start'
      on Click: SetBit("Data_Tank1_Heating_Cmd_StartMan")
   Button "Button_23" at 197,311 size 77x32; TextOff 'Stop'
      on Click: SetBit("Data_Tank1_Heating_Cmd_StopMan")
   Button "Button_24" at 357,311 size 77x32; TextOff 'Rsume'
      on Click: SetBit("Data_Tank1_Heating_Cmd_ResumeMan")
   Button "Button_25" at 277,311 size 77x32; TextOff 'Pause'
      on Click: SetBit("Data_Tank1_Heating_Cmd_PauseMan")
   Circle "Circle_16" at 394,225 size 20x20
      Appearance <- "Data_Tank1_Heating_State_Done"
   Button "Button_26" at 457,176 size 76x81; TextOff 'Text'
      on Click: ActivateScreen("MainScr", 0)
   Button "Button_9" at 121,260 size 77x32; TextOff 'Aut'
      on Click: SetBit("Data_Tank1_Mixer_Cmd_AutCtrl")
   TextField "Text field_12" at 119,191 size 83x23; Text 'Automat'
   TextField "Text field_13" at 119,209 size 70x23; Text 'Manual'
   TextField "Text field_14" at 119,232 size 79x23; Text 'Running'
   Button "Button_10" at 200,260 size 77x32; TextOff 'Man'
      on Click: SetBit("Data_Tank1_Mixer_Cmd_ManCtrl")
   Button "Button_11" at 121,293 size 77x32; TextOff 'Start'
      on Click: SetBit("Data_Tank1_Mixer_Cmd_TurnOnMan")
   Button "Button_12" at 200,293 size 77x32; TextOff 'Stop'
      on Click: SetBit("Data_Tank1_Mixer_Cmd_TurnOffMan")
   TextField "Text field_16" at 662,99 size 77x27; Text 'Phases'
   Button "Button_15" at 617,148 size 171x29; TextOff 'Menu filling'
      on Click: ActivateScreen("Filling", 0)
   TextField "Text field_17" at 668,124 size 61x23; Text 'Filling'
   SymbolicIOField "Symbolic I/O field_2" at 617,179 size 171x32; TextOn '1'; TextOff '0'; TextList "Phases"
      ProcessValue <- "Data_Tank1_Filling_State_Stateint"
   Button "Button_16" at 617,236 size 171x29; TextOff 'Menu draining'
      on Click: ActivateScreen("Draining", 0)
   TextField "Text field_18" at 660,213 size 82x23; Text 'Draining'
   SymbolicIOField "Symbolic I/O field_3" at 617,267 size 171x32; TextOn '1'; TextOff '0'; TextList "Phases"
      ProcessValue <- "Data_Tank1_Draining_State_StateInt"
   Button "Button_17" at 617,324 size 171x29; TextOff 'Menu mixing'
      on Click: ActivateScreen("Mixing", 0)
   TextField "Text field_19" at 669,301 size 65x23; Text 'Mixing'
   SymbolicIOField "Symbolic I/O field_4" at 617,355 size 171x32; TextOn '1'; TextOff '0'; TextList "Phases"
      ProcessValue <- "Data_Tank1_Mixing_State_StateInt"
   Button "Button_18" at 617,412 size 171x29; TextOff 'Menu heating'
      on Click: ActivateScreen("Heating", 0)
   TextField "Text field_20" at 665,390 size 76x23; Text 'Heating'
   SymbolicIOField "Symbolic I/O field_5" at 617,443 size 171x32; TextOn '1'; TextOff '0'; TextList "Phases"
      ProcessValue <- "Data_Tank1_Heating_State_StateInt"
   TextField "Text field_22" at 352,198 size 83x23; Text 'Automat'
   TextField "Text field_23" at 352,216 size 70x23; Text 'Manual'
   TextField "Text field_24" at 356,238 size 157x23; Text 'Manual heat pwr'
   IOField "I/O field_3" at 381,259 size 96x32; FormatPattern 999.9; Unit  %
      ProcessValue <- "Data_Tank1_Heater_Param_HeatingPowerManual"
   TextField "Text field_25" at 356,290 size 160x23; Text 'Req temperature'
   IOField "I/O field_4" at 381,311 size 96x32; FormatPattern 999.9; Unit  °C
      ProcessValue <- "Data_Tank1_Heating_Param_ReqTemp"
   Circle "Circle_9" at 236,192 size 20x20
      Appearance <- "Data_Tank1_Mixer_State_AutCtrl"
   Circle "Circle_10" at 236,212 size 20x20
      Appearance <- "Data_Tank1_Mixer_State_ManCtrl"
   Circle "Circle_12" at 236,236 size 20x20
      Appearance <- "Data_Tank1_Mixer_State_Run"
   Circle "Circle_11" at 469,199 size 20x20
      Appearance <- "Data_Tank1_Heating_Cmd_AutCtrl"
   Circle "Circle_13" at 469,219 size 20x20
      Appearance <- "Data_Tank1_Heating_Cmd_ManCtrl"

screen "Mixing" 800x480
   TextField "Text field_26" at 216,145 size 194x23; Text 'Mixing phase control'
   TextField "Text field_27" at 112,179 size 83x23; Text 'Automat'
   TextField "Text field_28" at 112,197 size 70x23; Text 'Manual'
   TextField "Text field_29" at 273,188 size 51x23; Text 'Done'
   GraphicView "Graphic view_1" at 455,140 size 75x74; Picture "exit-png-cancel-cross-exit-remove-icon-512"
   Button "Button_19" at 113,227 size 77x32; TextOff 'Aut'
      on Click: SetBit("Data_Tank1_Mixing_Cmd_AutCtrl")
   Button "Button_20" at 193,227 size 77x32; TextOff 'Man'
      on Click: SetBit("Data_Tank1_Mixing_Cmd_ManCtrl")
   Circle "Circle_14" at 229,181 size 20x20
      Appearance <- "Data_Tank1_Mixing_State_AutCtrl"
   Circle "Circle_15" at 229,201 size 20x20
      Appearance <- "Data_Tank1_Mixing_State_ManCtrl"
   Button "Button_21" at 274,227 size 157x32; TextOff 'Reset done'
      on Click: SetBit("Data_Tank1_Mixing_Cmd_ResetDone")
   Button "Button_22" at 113,277 size 77x32; TextOff 'Start'
      on Click: SetBit("Data_Tank1_Mixing_Cmd_StartMan")
   Button "Button_23" at 193,276 size 77x32; TextOff 'Stop'
      on Click: SetBit("Data_Tank1_Mixing_Cmd_StopMan")
   Button "Button_24" at 353,276 size 77x32; TextOff 'Rsume'
      on Click: SetBit("Data_Tank1_Mixing_Cmd_ResumeMan")
   Button "Button_25" at 273,276 size 77x32; TextOff 'Pause'
      on Click: SetBit("Data_Tank1_Mixing_Cmd_PauseMan")
   Circle "Circle_16" at 390,190 size 20x20
      Appearance <- "Data_Tank1_Mixing_State_Done"
   Button "Button_26" at 451,141 size 76x81; TextOff 'Text'
      on Click: ActivateScreen("MainScr", 0)
   Button "Button_9" at 117,272 size 77x32; TextOff 'Aut'
      on Click: SetBit("Data_Tank1_Mixer_Cmd_AutCtrl")
   TextField "Text field_11" at 164,178 size 56x23; Text 'Mixer'
   TextField "Text field_12" at 115,203 size 83x23; Text 'Automat'
   TextField "Text field_13" at 115,221 size 70x23; Text 'Manual'
   TextField "Text field_14" at 115,244 size 79x23; Text 'Running'
   Button "Button_10" at 196,272 size 77x32; TextOff 'Man'
      on Click: SetBit("Data_Tank1_Mixer_Cmd_ManCtrl")
   TextField "Text field_16" at 662,99 size 77x27; Text 'Phases'
   Button "Button_15" at 617,148 size 171x29; TextOff 'Menu filling'
      on Click: ActivateScreen("Filling", 0)
   TextField "Text field_17" at 668,124 size 61x23; Text 'Filling'
   SymbolicIOField "Symbolic I/O field_2" at 617,179 size 171x32; TextOn '1'; TextOff '0'; TextList "Phases"
      ProcessValue <- "Data_Tank1_Filling_State_Stateint"
   Button "Button_16" at 617,236 size 171x29; TextOff 'Menu draining'
      on Click: ActivateScreen("Draining", 0)
   TextField "Text field_18" at 660,213 size 82x23; Text 'Draining'
   SymbolicIOField "Symbolic I/O field_3" at 617,267 size 171x32; TextOn '1'; TextOff '0'; TextList "Phases"
      ProcessValue <- "Data_Tank1_Draining_State_StateInt"
   Button "Button_17" at 617,324 size 171x29; TextOff 'Menu mixing'
      on Click: ActivateScreen("Mixing", 0)
   TextField "Text field_19" at 669,301 size 65x23; Text 'Mixing'
   SymbolicIOField "Symbolic I/O field_4" at 617,355 size 171x32; TextOn '1'; TextOff '0'; TextList "Phases"
      ProcessValue <- "Data_Tank1_Mixing_State_StateInt"
   Button "Button_18" at 617,412 size 171x29; TextOff 'Menu heating'
      on Click: ActivateScreen("Heating", 0)
   TextField "Text field_20" at 665,390 size 76x23; Text 'Heating'
   SymbolicIOField "Symbolic I/O field_5" at 617,443 size 171x32; TextOn '1'; TextOff '0'; TextList "Phases"
      ProcessValue <- "Data_Tank1_Heating_State_StateInt"
   TextField "Text field_21" at 357,185 size 156x23; Text 'Heating element'
   TextField "Text field_22" at 348,210 size 83x23; Text 'Automat'
   TextField "Text field_23" at 348,228 size 70x23; Text 'Manual'
   TextField "Text field_24" at 352,250 size 157x23; Text 'Manual heat pwr'
   IOField "I/O field_3" at 377,271 size 96x32; FormatPattern 999.9; Unit  %
      ProcessValue <- "Data_Tank1_Heater_Param_HeatingPowerManual"
   TextField "Text field_25" at 352,302 size 160x23; Text 'Req temperature'
   Circle "Circle_9" at 232,204 size 20x20
      Appearance <- "Data_Tank1_Mixer_State_AutCtrl"
   Circle "Circle_10" at 232,224 size 20x20
      Appearance <- "Data_Tank1_Mixer_State_ManCtrl"
   Circle "Circle_12" at 232,248 size 20x20
      Appearance <- "Data_Tank1_Mixer_State_Run"
   Circle "Circle_11" at 465,211 size 20x20
      Appearance <- "Data_Tank1_Heating_Cmd_AutCtrl"
   Circle "Circle_13" at 465,231 size 20x20
      Appearance <- "Data_Tank1_Heating_Cmd_ManCtrl"
   TextField "Text field_30" at 357,179 size 156x23; Text 'Heating element'
   TextField "Text field_31" at 348,204 size 83x23; Text 'Automat'
   TextField "Text field_32" at 348,222 size 70x23; Text 'Manual'
   TextField "Text field_33" at 352,244 size 157x23; Text 'Manual heat pwr'
   Circle "Circle_17" at 465,205 size 20x20
      Appearance <- "Data_Tank1_Heater_State_AutCtrl"
   Circle "Circle_18" at 465,225 size 20x20
      Appearance <- "Data_Tank1_Heater_State_ManCtrl"
   IOField "I/O field_4" at 377,265 size 96x32; FormatPattern 999.9; Unit  %
      ProcessValue <- "Data_Tank1_Heater_Param_HeatingPowerManual"

screen "Filling" 800x480
   Button "Button_19" at 100,212 size 77x32; TextOff 'Aut'
      on Click: SetBit("Data_Tank1_Filling_Cmd_AutCtrl")
   TextField "Text field_26" at 203,131 size 190x23; Text 'Filling phase control'
   TextField "Text field_27" at 99,165 size 83x23; Text 'Automat'
   TextField "Text field_28" at 99,183 size 70x23; Text 'Manual'
   Button "Button_20" at 180,212 size 77x32; TextOff 'Man'
      on Click: SetBit("Data_Tank1_Filling_Cmd_ManCtrl")
   Circle "Circle_14" at 216,166 size 20x20
      Appearance <- "Data_Tank1_Filling_State_AutCtrl"
   Circle "Circle_15" at 216,186 size 20x20
      Appearance <- "Data_Tank1_Filling_State_ManCtrl"
   Button "Button_21" at 261,212 size 157x32; TextOff 'Reset done'
      on Click: SetBit("Data_Tank1_Filling_Cmd_ResetDone")
   Button "Button_22" at 100,262 size 77x32; TextOff 'Start'
      on Click: SetBit("Data_Tank1_Filling_Cmd_StartMan")
   Button "Button_23" at 180,261 size 77x32; TextOff 'Stop'
      on Click: SetBit("Data_Tank1_Filling_Cmd_StopMan")
   Button "Button_24" at 340,261 size 77x32; TextOff 'Rsume'
      on Click: SetBit("Data_Tank1_Filling_Cmd_ResumeMan")
   Button "Button_25" at 260,261 size 77x32; TextOff 'Pause'
      on Click: SetBit("Data_Tank1_Filling_Cmd_PauseMan")
   TextField "Text field_29" at 260,174 size 51x23; Text 'Done'
   Circle "Circle_16" at 377,175 size 20x20
      Appearance <- "Data_Tank1_Filling_State_Done"
   GraphicView "Graphic view_1" at 442,126 size 75x74; Picture "exit-png-cancel-cross-exit-remove-icon-512"
   Button "Button_26" at 437,128 size 76x81; TextOff 'Text'
      on Click: ActivateScreen("MainScr", 0)
   TextField "Text field_16" at 662,99 size 77x27; Text 'Phases'
   Button "Button_15" at 617,148 size 171x29; TextOff 'Menu filling'
      on Click: ActivateScreen("Filling", 0)
   TextField "Text field_17" at 668,124 size 61x23; Text 'Filling'
   SymbolicIOField "Symbolic I/O field_2" at 617,179 size 171x32; TextOn '1'; TextOff '0'; TextList "Phases"
      ProcessValue <- "Data_Tank1_Filling_State_Stateint"
   Button "Button_16" at 617,236 size 171x29; TextOff 'Menu draining'
      on Click: ActivateScreen("Draining", 0)
   TextField "Text field_18" at 660,213 size 82x23; Text 'Draining'
   SymbolicIOField "Symbolic I/O field_3" at 617,267 size 171x32; TextOn '1'; TextOff '0'; TextList "Phases"
      ProcessValue <- "Data_Tank1_Draining_State_StateInt"
   Button "Button_17" at 617,324 size 171x29; TextOff 'Menu mixing'
      on Click: ActivateScreen("Mixing", 0)
   TextField "Text field_19" at 669,301 size 65x23; Text 'Mixing'
   SymbolicIOField "Symbolic I/O field_4" at 617,355 size 171x32; TextOn '1'; TextOff '0'; TextList "Phases"
      ProcessValue <- "Data_Tank1_Mixing_State_StateInt"
   Button "Button_18" at 617,412 size 171x29; TextOff 'Menu heating'
      on Click: ActivateScreen("Heating", 0)
   TextField "Text field_20" at 665,390 size 76x23; Text 'Heating'
   SymbolicIOField "Symbolic I/O field_5" at 617,443 size 171x32; TextOn '1'; TextOff '0'; TextList "Phases"
      ProcessValue <- "Data_Tank1_Heating_State_StateInt"

screen "Draining" 800x480
   Button "Button_25" at 266,295 size 77x32; TextOff 'Pause'
      on Click: SetBit("Data_Tank1_Draining_Cmd_PauseMan")
   Button "Button_23" at 186,295 size 77x32; TextOff 'Stop'
      on Click: SetBit("Data_Tank1_Draining_Cmd_StopMan")
   Button "Button_22" at 106,296 size 77x32; TextOff 'Start'
      on Click: SetBit("Data_Tank1_Draining_Cmd_StartMan")
   Button "Button_19" at 106,246 size 77x32; TextOff 'Aut'
      on Click: SetBit("Data_Tank1_Draining_Cmd_AutCtrl")
   Button "Button_20" at 186,246 size 77x32; TextOff 'Man'
      on Click: SetBit("Data_Tank1_Draining_Cmd_ManCtrl")
   Button "Button_21" at 267,246 size 157x32; TextOff 'Reset done'
      on Click: SetBit("Data_Tank1_Draining_Cmd_ResetDone")
   TextField "Text field_28" at 105,218 size 70x23; Text 'Manual'
   TextField "Text field_27" at 105,200 size 83x23; Text 'Automat'
   Circle "Circle_16" at 383,209 size 20x20
      Appearance <- "Data_Tank1_Draining_State_Done"
   Circle "Circle_15" at 222,220 size 20x20
      Appearance <- "Data_Tank1_Draining_State_ManCtrl"
   Circle "Circle_14" at 222,200 size 20x20
      Appearance <- "Data_Tank1_Draining_State_AutCtrl"
   TextField "Text field_26" at 209,166 size 211x23; Text 'Draining phase control'
   TextField "Text field_29" at 266,209 size 51x23; Text 'Done'
   Button "Button_24" at 346,295 size 77x32; TextOff 'Rsume'
      on Click: SetBit("Data_Tank1_Draining_Cmd_ResumeMan")
   GraphicView "Graphic view_1" at 448,162 size 75x74; Picture "exit-png-cancel-cross-exit-remove-icon-512"
   Button "Button_26" at 447,166 size 76x81; TextOff 'Text'
      on Click: ActivateScreen("MainScr", 0)
   TextField "Text field_16" at 662,99 size 77x27; Text 'Phases'
   Button "Button_15" at 617,148 size 171x29; TextOff 'Menu filling'
      on Click: ActivateScreen("Filling", 0)
   TextField "Text field_17" at 668,124 size 61x23; Text 'Filling'
   SymbolicIOField "Symbolic I/O field_2" at 617,179 size 171x32; TextOn '1'; TextOff '0'; TextList "Phases"
      ProcessValue <- "Data_Tank1_Filling_State_Stateint"
   Button "Button_16" at 617,236 size 171x29; TextOff 'Menu draining'
      on Click: ActivateScreen("Draining", 0)
   TextField "Text field_18" at 660,213 size 82x23; Text 'Draining'
   SymbolicIOField "Symbolic I/O field_3" at 617,267 size 171x32; TextOn '1'; TextOff '0'; TextList "Phases"
      ProcessValue <- "Data_Tank1_Draining_State_StateInt"
   Button "Button_17" at 617,324 size 171x29; TextOff 'Menu mixing'
      on Click: ActivateScreen("Mixing", 0)
   TextField "Text field_19" at 669,301 size 65x23; Text 'Mixing'
   SymbolicIOField "Symbolic I/O field_4" at 617,355 size 171x32; TextOn '1'; TextOff '0'; TextList "Phases"
      ProcessValue <- "Data_Tank1_Mixing_State_StateInt"
   Button "Button_18" at 617,412 size 171x29; TextOff 'Menu heating'
      on Click: ActivateScreen("Heating", 0)
   TextField "Text field_20" at 665,390 size 76x23; Text 'Heating'
   SymbolicIOField "Symbolic I/O field_5" at 617,443 size 171x32; TextOn '1'; TextOff '0'; TextList "Phases"
      ProcessValue <- "Data_Tank1_Heating_State_StateInt"

screen "Parameters" 800x480
   Button "Button_19" at 659,404 size 130x66; TextOff 'Main screen'
      on Click: ActivateScreen("MainScr", 0)
   TextField "Text field_24" at 65,77 size 83x23; Text 'Fill level'
   IOField "I/O field_3" at 222,77 size 96x32; FormatPattern 9.9; Unit  m
      ProcessValue <- "Data_Tank1_Filling_Param_FillLevel"
   TextField "Text field_1" at 65,121 size 104x23; Text 'Drain level'
   IOField "I/O field_1" at 222,120 size 96x32; FormatPattern 9.9; Unit  m
      ProcessValue <- "Data_Tank1_Draining_Param_DrainLevel"
   TextField "Text field_2" at 65,166 size 112x23; Text 'Mixing time'
   IOField "I/O field_2" at 222,166 size 96x32; FormatPattern 99; Unit  s
      ProcessValue <- "Data_Tank1_Mixing_Param_TimeSec"
   TextField "Text field_3" at 65,214 size 163x23; Text 'Heating set point'
   IOField "I/O field_4" at 222,212 size 96x32; FormatPattern 99; Unit  °C
      ProcessValue <- "Data_Tank1_Heater_Param_HeatingSetPointAutomat"
*)